// TwinCAT 3 PLC project Main
// ProgramVersion: 3.1.4026.19
// libraries:
//   Tc2_EtherCAT, * (Beckhoff Automation GmbH)
//   Tc2_MC2, * (Beckhoff Automation GmbH)
//   Tc2_Standard, * (Beckhoff Automation GmbH)
//   Tc2_System, * (Beckhoff Automation GmbH)
//   Tc2_Utilities, * (Beckhoff Automation GmbH)
//   Tc3_Database, * (Beckhoff Automation GmbH)
//   Tc3_EventLogger, * (Beckhoff Automation GmbH)
//   Tc3_JsonXml, * (Beckhoff Automation GmbH)
//   Tc3_Module, * (Beckhoff Automation GmbH)
// project tree:
//   DUTs/ ActionMode.TcDUT, MachineState.TcDUT, Sub_Step.TcDUT, TestAction.TcDUT
//   DUTs/IO模組/ IO_In16.TcDUT, IO_Out16.TcDUT
//   DUTs/Jog_STRUCT/ Jog_Laser_Group.TcDUT, Jog_Fx_Group.TcDUT
//   DUTs/加工資料結構/材料加工資訊結構/ tsSteelData.TcDUT
//   DUTs/加工資料結構/工單結構/ WorkOrder_Data.TcDUT
//   DUTs/加工資料結構/雷射加工參數/ LaserParameter_Data.TcDUT
//   DUTs/加工資料結構/雷射加工資料/ LaserProcess_Data.TcDUT
//   DUTs/座標/ XYZ_Point.TcDUT
//   GVLs/ Axis.TcGVL, GrobelVariable.TcGVL, Hmi.TcGVL, Hmi_Web.TcGVL, MaCfg.TcGVL, IO.TcGVL, PosC.TcGVL, ProjectData.TcGVL, RecipeManager.TcRMO (not stored), Safety.TcGVL, SensorTest.TcGVL, AxisTest.TcGVL, SpdC.TcGVL
//   MSG/訊息列表/ MsgBuff.TcGVL
//   MSG/訊息格式/ MsgLevel.TcDUT, MsgStruct.TcDUT, MsgStruct_RAW.TcDUT
//   MSG/通知訊息/ MsgMain.TcPOU, MsgPush.TcPOU, uuidv7_g.TcPOU
//   / PlcTask.TcTTO
//   POUs/ MAIN.TcPOU
//   POUs/功能塊/ ErrorCodeConver.TcPOU, pMsg.TcPOU, RW_Config.TcPOU
//   POUs/功能塊/EtherCat相關/ EtherCat_Driver_Reset.TcPOU, GetEtherSta.TcPOU, EtherCAT_Status.TcPOU
//   POUs/功能塊/Stober驅動/ ReadStoberError.TcPOU, StoberErrorStr.TcPOU
//   POUs/功能塊/字串處理功能塊/字串填充/ FILLSTRING.TcPOU
//   POUs/功能塊/字串處理功能塊/浮點轉字串控制去小數點/ Real2String.TcPOU
//   POUs/功能塊/字串處理功能塊/字串記憶/ WStrMem.TcPOU
//   POUs/功能塊/字串處理功能塊/字串連接/ StrConcat.TcPOU, WStrConcat.TcPOU
//   POUs/功能塊/資料庫 Postgre相關/ ReadSQLData.TcPOU
//   POUs/功能塊/資料庫 Postgre相關/相關結構/取得範圍內的加工資料/ SQL_Get_Payload_Struct.TcDUT
//   POUs/功能塊/資料庫 Postgre相關/相關結構/取得X點/ SQL_GetPosX_Struct.TcDUT
//   POUs/功能塊/資料庫 Postgre相關/相關結構/寫入起始時間/ Payload_Write_Time.TcDUT
//   POUs/功能塊/資料庫 Postgre相關/記錄用/滾輪誤差紀錄/ FxErrPos.TcPOU (not stored), FxErrPos_Struct.TcDUT (not stored)
//   POUs/功能塊/資料庫 Postgre相關/記錄用/程式紀錄/ StepLog_Struct.TcDUT, Step_Log.TcPOU, Step_Log_Clear.TcPOU
//   POUs/動作流程控制/AxisGroup功能塊/ GroupA.TcPOU, GroupB.TcPOU, GroupC.TcPOU, GroupD.TcPOU, GroupFx.TcPOU
//   POUs/動作流程控制/外部輸送滾輪/ ExpConver.TcPOU
//   POUs/安全控制/ MaBaseState.TcPOU
//   POUs/硬體控制/其他控制/按鈕燈/ Button.TcPOU
//   POUs/硬體控制/其他控制/螢幕旋轉/ TurnMonitor.TcPOU
//   POUs/硬體控制/手搖輪/ Jog_MPG.TcPOU
//   POUs/硬體控制/測距感應器/ I_DisSensor.TcIO, OMH555_Decoder.TcPOU, DT80_Decoder.TcPOU, Sensor.TcPOU
//   POUs/硬體控制/軸/ AxisAction.TcPOU, AxisBase.TcPOU, I_Axis.TcIO, MultipleAxisBase.TcPOU, AxisFx.TcPOU
//   POUs/硬體控制/其他控制/三色燈/ LightTower.TcPOU
//   POUs/動作流程控制/ AutoMain.TcPOU
//   POUs/動作流程控制/人機資料轉換/ WebHmi.TcPOU
//   POUs/動作流程控制/測試功能/ Sql_TestData.TcDUT, Sql_TestWriteData.TcDUT, TestActionPou.TcPOU
// real-time tasks:
//   TASK Main_IO_Task: cycle T#2ms, priority 6, ADS port 353
//   TASK PlcTask: cycle T#10ms, priority 14, ADS port 350
//   TASK Conveyor: cycle T#10ms, priority 22, ADS port 355
// motion (NC):
//   TASK NC-Task 1 SAF: cycle T#2ms, priority 4, ADS port 501
//   TASK NC-Task 1 SVB: cycle T#10ms, priority 8, ADS port 511
//   AXIS FX1 (id 1)
//     Dynamic: Acceleration=300, Deceleration=300, Jerk=2000
//     Velo: SlowManual=30, FastManual=300
//     PositionAreaControl: Enable=false
//     OtherSettings: AllowMotionCmdToSlave=true
//     encoder EncType=19
//       EncPara: ScaleFactorNumerator=6.574203208, ScaleFactorDenominator=1048576, Inverse=true, MaxCount=#xffffffff
//     encoder EncId=129, EncType=4
//       EncPara: MaxCount=#xffffffff
//         Inc: RefMode=2
//     encoder EncId=145, EncType=4
//       EncPara: MaxCount=#xffffffff
//         Inc: RefMode=2
//     drive DrvType=16
//       DrvPara: Inverse=true, MaxCount=#xffffffff, DriveControlDWord=#x00020100
//         Analog: TorqueSetpointScale=10, ScaleFactorActTorque=0.1
//         TimeComp: TaskDelayCycles=1
//     controller CtrType=1
//       CtrPara: PriorControlFactor=1
//         PosDiffControl: Enable=false
//         Observer: BandWidth=20
//   AXIS FX2 (id 2)
//     Dynamic: Acceleration=200, Deceleration=200, Jerk=100
//     Velo: FastManual=400, Maximum=600
//     OtherSettings: AllowMotionCmdToSlave=true
//     encoder EncType=19
//       EncPara: ScaleFactorNumerator=6.574203208, ScaleFactorDenominator=1048576, Inverse=true, MaxCount=#xffffffff
//     drive DrvType=16
//       DrvPara: Inverse=true, MaxCount=#xffffffff, DriveControlDWord=#x00020100
//         Analog: TorqueSetpointScale=10, ScaleFactorActTorque=0.1
//         TimeComp: TaskDelayCycles=1
//     controller CtrType=1
//       CtrPara: PriorControlFactor=1
//         Observer: BandWidth=20
//   AXIS AX (id 3)
//     Dynamic: AccelerationMaximum=1000, DecelerationMaximum=1000, Acceleration=1000, Deceleration=1000, Jerk=10000
//     Velo: SlowManual=10, FastManual=50, Maximum=545
//     OtherSettings: AllowMotionCmdToSlave=true, PulseDistancePos=1, PulseDistanceNeg=1
//     encoder EncType=19
//       EncPara: ScaleFactorNumerator=10.6657070589373, ScaleFactorDenominator=1048576, MaxCount=#xffffffff, ReferenceSystem=1
//         SoftEndMinControl: Range=-2
//         SoftEndMaxControl: Range=337
//     drive DrvType=16
//       DrvPara: MaxCount=#xffffffff, DriveControlDWord=#x00020100
//         Analog: VeloReferenz=590, TorqueSetpointScale=10, ScaleFactorActTorque=0.1
//         TimeComp: TaskDelayCycles=1
//     controller CtrType=1
//       CtrPara: PriorControlFactor=1
//         Observer: BandWidth=20
//   AXIS AY (id 4)
//     Dynamic: Acceleration=1000, Deceleration=1000, Jerk=10000
//     Velo: SlowManual=10, FastManual=50, Maximum=545
//     OtherSettings: AllowMotionCmdToSlave=true
//     encoder EncType=19
//       EncPara: ScaleFactorNumerator=10.5986464258042, ScaleFactorDenominator=1048576, Offset=-3.99996967702935, MaxCount=#xffffffff, ReferenceSystem=1
//         SoftEndMinControl: Range=-2
//         SoftEndMaxControl: Range=635.996398925781
//     drive DrvType=16
//       DrvPara: MaxCount=#xffffffff, DriveControlDWord=#x00020100
//         Analog: VeloReferenz=590, TorqueSetpointScale=10, ScaleFactorActTorque=0.1
//         TimeComp: TaskDelayCycles=1
//     controller CtrType=1
//       CtrPara: PriorControlFactor=1
//         Observer: BandWidth=20
//   AXIS AZ1 (id 5)
//     Dynamic: Acceleration=1000, Deceleration=1000, Jerk=10000
//     Velo: SlowManual=10, FastManual=50, Maximum=545
//     OtherSettings: AllowMotionCmdToSlave=true
//     encoder EncType=19
//       EncPara: ScaleFactorNumerator=10.6657070589373, ScaleFactorDenominator=1048576, Inverse=true, MaxCount=#xffffffff, ReferenceSystem=1
//         SoftEndMinControl: Range=-2
//         SoftEndMaxControl: Range=316.997497558594
//     drive DrvType=16
//       DrvPara: Inverse=true, MaxCount=#xffffffff, DriveControlDWord=#x00020100
//         Analog: VeloReferenz=590, TorqueSetpointScale=10, ScaleFactorActTorque=0.1
//         TimeComp: TaskDelayCycles=1
//     controller CtrType=1
//       CtrPara: PriorControlFactor=1
//         Observer: BandWidth=20
//   AXIS AZ2 (id 6)
//     Dynamic: Acceleration=1000, Deceleration=1000, Jerk=10000
//     Velo: SlowManual=10, FastManual=50, Maximum=545
//     OtherSettings: AllowMotionCmdToSlave=true
//     encoder EncType=19
//       EncPara: ScaleFactorNumerator=10.6657070589373, ScaleFactorDenominator=1048576, MaxCount=#xffffffff, ReferenceSystem=1
//     drive DrvType=16
//       DrvPara: MaxCount=#xffffffff, DriveControlDWord=#x00020100
//         Analog: VeloReferenz=590, TorqueSetpointScale=10, ScaleFactorActTorque=0.1
//         TimeComp: TaskDelayCycles=1
//     controller CtrType=1
//       CtrPara: PriorControlFactor=1
//         Observer: BandWidth=20
//   AXIS BX (id 7)
//     Dynamic: Acceleration=1000, Deceleration=1000, Jerk=10000
//     Velo: SlowManual=10, FastManual=50, Maximum=545
//     OtherSettings: AllowMotionCmdToSlave=true
//     encoder EncType=19
//       EncPara: ScaleFactorNumerator=10.6657070589373, ScaleFactorDenominator=1048576, Inverse=true, MaxCount=#xffffffff, ReferenceSystem=1
//         SoftEndMinControl: Range=10
//         SoftEndMaxControl: Range=400
//         Inc: RefSoftSyncMask=#xffffffff
//     drive DrvType=16
//       DrvPara: Inverse=true, MaxCount=#xffffffff, DriveControlDWord=#x00020100
//         Analog: VeloReferenz=590, TorqueSetpointScale=10, ScaleFactorActTorque=0.1
//         TimeComp: TaskDelayCycles=1
//     controller CtrType=1
//       CtrPara: PriorControlFactor=1
//         Observer: BandWidth=20
//   AXIS BY1 (id 8)
//     Dynamic: Acceleration=1000, Deceleration=1000, Jerk=10000
//     Velo: SlowManual=10, FastManual=50, Maximum=545
//     BacklashCompensation: Range=0.05
//     OtherSettings: AllowMotionCmdToSlave=true
//     encoder EncType=19
//       EncPara: ScaleFactorNumerator=10.6657070589373, ScaleFactorDenominator=1048576, Inverse=true, MaxCount=#xffffffff, ReferenceSystem=1
//         SoftEndMinControl: Range=-2
//         SoftEndMaxControl: Range=1405
//     drive DrvType=16
//       DrvPara: Inverse=true, MaxCount=#xffffffff, DriveControlDWord=#x00020100
//         Analog: VeloReferenz=590, TorqueSetpointScale=10, ScaleFactorActTorque=0.1
//         TimeComp: TaskDelayCycles=1
//     controller CtrType=1
//       CtrPara: PriorControlFactor=1
//         Observer: BandWidth=20
//   AXIS BY2 (id 9)
//     Dynamic: Acceleration=1000, Deceleration=1000, Jerk=10000
//     Velo: SlowManual=10, FastManual=50, Maximum=545
//     OtherSettings: ErrorReactionDelay=0.05, AllowMotionCmdToSlave=true
//     encoder EncType=19
//       EncPara: ScaleFactorNumerator=10.6657070589373, ScaleFactorDenominator=1048576, MaxCount=#xffffffff, ReferenceSystem=1
//     drive DrvType=16
//       DrvPara: MaxCount=#xffffffff, DriveControlDWord=#x00020100
//         Analog: VeloReferenz=590, TorqueSetpointScale=10, ScaleFactorActTorque=0.1
//         TimeComp: TaskDelayCycles=1
//     controller CtrType=1
//       CtrPara: PriorControlFactor=1
//         Observer: BandWidth=20
//   AXIS BZ (id 10)
//     Dynamic: Acceleration=1000, Deceleration=1000, Jerk=10000
//     Velo: SlowManual=10, FastManual=50, Maximum=545
//     OtherSettings: AllowMotionCmdToSlave=true
//     encoder EncType=19
//       EncPara: ScaleFactorNumerator=10.6657070589373, ScaleFactorDenominator=1048576, Inverse=true, MaxCount=#xffffffff, ReferenceSystem=1
//         SoftEndMinControl: Range=-2
//         SoftEndMaxControl: Range=601.999633789063
//     drive DrvType=16
//       DrvPara: Inverse=true, MaxCount=#xffffffff, DriveControlDWord=#x00020100
//         Analog: VeloReferenz=590, TorqueSetpointScale=10, ScaleFactorActTorque=0.1
//         TimeComp: TaskDelayCycles=1
//     controller CtrType=1
//       CtrPara: PriorControlFactor=1
//         Observer: BandWidth=20
//   AXIS CX (id 11)
//     Dynamic: Acceleration=1000, Deceleration=1000, Jerk=10000
//     Velo: SlowManual=10, FastManual=50, Maximum=545
//     OtherSettings: AllowMotionCmdToSlave=true
//     encoder EncType=19
//       EncPara: ScaleFactorNumerator=10.6657070589373, ScaleFactorDenominator=1048576, Inverse=true, MaxCount=#xffffffff, ReferenceSystem=1
//         SoftEndMinControl: Range=-2
//         SoftEndMaxControl: Range=317.003509521484
//     drive DrvType=16
//       DrvPara: Inverse=true, MaxCount=#xffffffff, DriveControlDWord=#x00020100
//         Analog: VeloReferenz=590, TorqueSetpointScale=10, ScaleFactorActTorque=0.1
//         TimeComp: TaskDelayCycles=1
//     controller CtrType=1
//       CtrPara: PriorControlFactor=1
//         Observer: BandWidth=20
//   AXIS CY (id 12)
//     Dynamic: Acceleration=1000, Deceleration=1000, Jerk=10000
//     Velo: SlowManual=10, FastManual=50, Maximum=545
//     OtherSettings: AllowMotionCmdToSlave=true
//     encoder EncType=19
//       EncPara: ScaleFactorNumerator=10.6657070589373, ScaleFactorDenominator=1048576, Inverse=true, MaxCount=#xffffffff, ReferenceSystem=1
//         SoftEndMinControl: Range=-2
//         SoftEndMaxControl: Range=623.000061035156
//     drive DrvType=16
//       DrvPara: Inverse=true, MaxCount=#xffffffff, DriveControlDWord=#x00020100
//         Analog: VeloReferenz=590, TorqueSetpointScale=10, ScaleFactorActTorque=0.1
//         TimeComp: TaskDelayCycles=1
//     controller CtrType=1
//       CtrPara: PriorControlFactor=1
//         Observer: BandWidth=20
//   AXIS CZ1 (id 13)
//     Dynamic: Acceleration=1000, Deceleration=1000, Jerk=10000
//     Velo: SlowManual=10, FastManual=50, Maximum=545
//     OtherSettings: AllowMotionCmdToSlave=true
//     encoder EncType=19
//       EncPara: ScaleFactorNumerator=10.6657070589373, ScaleFactorDenominator=1048576, EncMode=3, MaxCount=#xffffffff, ReferenceSystem=1
//         SoftEndMinControl: Range=-2
//         SoftEndMaxControl: Range=1231.99340820313
//     drive DrvType=16
//       DrvPara: MaxCount=#xffffffff, DriveControlDWord=#x00020100
//         Analog: VeloReferenz=590, TorqueSetpointScale=10, ScaleFactorActTorque=0.1
//         TimeComp: TaskDelayCycles=1
//     controller CtrType=1
//       CtrPara: PriorControlFactor=1
//         Observer: BandWidth=20
//   AXIS CZ2 (id 14)
//     Dynamic: Acceleration=1000, Deceleration=1000, Jerk=10000
//     Velo: SlowManual=10, FastManual=50, Maximum=545
//     OtherSettings: AllowMotionCmdToSlave=true
//     encoder EncType=19
//       EncPara: ScaleFactorNumerator=10.6657070589373, ScaleFactorDenominator=1048576, Inverse=true, MaxCount=#xffffffff, ReferenceSystem=1
//     drive DrvType=16
//       DrvPara: Inverse=true, MaxCount=#xffffffff, DriveControlDWord=#x00020100
//         Analog: VeloReferenz=590, TorqueSetpointScale=10, ScaleFactorActTorque=0.1
//         TimeComp: TaskDelayCycles=1
//     controller CtrType=1
//       CtrPara: PriorControlFactor=1
//         Observer: BandWidth=20
//   AXIS DX (id 15)
//     Dynamic: Acceleration=1000, Deceleration=1000, Jerk=10000
//     Velo: SlowManual=10, FastManual=50, Maximum=545
//     OtherSettings: AllowMotionCmdToSlave=true
//     encoder EncType=19
//       EncPara: ScaleFactorNumerator=10.6657070589373, ScaleFactorDenominator=1048576, Offset=-2.99948538910209, Inverse=true, MaxCount=#xffffffff, ReferenceSystem=1
//         SoftEndMinControl: Range=-2
//         SoftEndMaxControl: Range=321.993438720703
//     drive DrvType=16
//       DrvPara: Inverse=true, MaxCount=#xffffffff, DriveControlDWord=#x00020100
//         Analog: VeloReferenz=590, TorqueSetpointScale=10, ScaleFactorActTorque=0.1
//         TimeComp: TaskDelayCycles=1
//     controller CtrType=1
//       CtrPara: PriorControlFactor=1
//         Observer: BandWidth=20
//   AXIS DY (id 16)
//     Dynamic: Acceleration=1000, Deceleration=1000, Jerk=10000
//     Velo: SlowManual=10, FastManual=50, Maximum=545
//     OtherSettings: AllowMotionCmdToSlave=true
//     encoder EncType=19
//       EncPara: ScaleFactorNumerator=10.6657070589373, ScaleFactorDenominator=1048576, MaxCount=#xffffffff, ReferenceSystem=1
//         SoftEndMinControl: Range=-2
//         SoftEndMaxControl: Range=1272
//     drive DrvType=16
//       DrvPara: MaxCount=#xffffffff, DriveControlDWord=#x00020100
//         Analog: VeloReferenz=590, TorqueSetpointScale=10, ScaleFactorActTorque=0.1
//         TimeComp: TaskDelayCycles=1
//     controller CtrType=1
//       CtrPara: PriorControlFactor=1
//         Observer: BandWidth=20
//   AXIS DZ (id 17)
//     Dynamic: Acceleration=1000, Deceleration=1000, Jerk=10000
//     Velo: SlowManual=10, FastManual=50, Maximum=545
//     OtherSettings: AllowMotionCmdToSlave=true
//     encoder EncType=19
//       EncPara: ScaleFactorNumerator=10.6657070589373, ScaleFactorDenominator=1048576, MaxCount=#xffffffff, ReferenceSystem=1
//         SoftEndMinControl: Range=-2
//         SoftEndMaxControl: Range=306.999847412109
//     drive DrvType=16
//       DrvPara: MaxCount=#xffffffff, DriveControlDWord=#x00020100
//         Analog: VeloReferenz=590, TorqueSetpointScale=10, ScaleFactorActTorque=0.1
//         TimeComp: TaskDelayCycles=1
//     controller CtrType=1
//       CtrPara: PriorControlFactor=1
//         Observer: BandWidth=20
//   AXIS MPG (id 18)
//     Dynamic: AccelerationMaximum=50, DecelerationMaximum=50
//     PositionAreaControl: Enable=false
//     TargetPosControl: Enable=false
//     OtherSettings: AllowMotionCmdToSlave=true
//     encoder EncType=4
//       EncPara: ScaleFactorNumerator=1, ModuloFactor=100, EncMode=3, MaxCount=#xffffffff
//         FilterTime: TPos=0.1, TVelo=0, TAcc=0
//         SoftEndMinControl: Range=-3
//         SoftEndMaxControl: Range=-99999
//         ActPosCorrection: Time=0.05
//     drive DrvType=5
//       Analog: VeloReferenz=500, TorqueSetpointScale=10, ScaleFactorActTorque=0.1
//       TimeComp: TaskDelayCycles=1
//     controller CtrType=1
//       CtrPara: PriorControlFactor=1
//         PosDiffControl: Enable=false
//         Observer: BandWidth=20
//   AXIS 轴 19 (id 19)
//     Dynamic: Acceleration=1000, Deceleration=1000, Jerk=5000
//     Velo: SlowManual=10, FastManual=120
//     OtherSettings: AllowMotionCmdToSlave=true
//     encoder EncType=19
//       EncPara: ScaleFactorNumerator=20, ScaleFactorDenominator=10000, ModuloFactor=20, MaxCount=#xffffffff
//     drive DrvType=16
//       DrvPara: MaxCount=#xffffffff, DriveControlDWord=#x00020100
//         Analog: TorqueSetpointScale=10, ScaleFactorActTorque=0.1
//         TimeComp: TaskDelayCycles=1
//     controller CtrType=1
//       CtrPara: PriorControlFactor=1
//         PosDiffControl: Enable=false
//         Observer: BandWidth=20
// I/O:
//   DEVICE Device 1 (EtherCAT), AmsNetId 0.0.0.0.2.1
//     Term 1 (EK1200) [EK1200-5000 EtherCAT Power supply (2A E-Bus)]
//       Term 2 (EL1409) [EL1409 16Ch. Dig. Input 24V, 3ms]
//       Term 3 (EL1409) [EL1409 16Ch. Dig. Input 24V, 3ms]
//       Term 4 (EL1409) [EL1409 16Ch. Dig. Input 24V, 3ms]
//       Term 5 (EL1409) [EL1409 16Ch. Dig. Input 24V, 3ms]
//       Term 6 (EL1409) [EL1409 16Ch. Dig. Input 24V, 3ms]
//       Term 7 (EL1409) [EL1409 16Ch. Dig. Input 24V, 3ms]
//       Term 8 (EL2409) [EL2409 16Ch. Dig. Output 24V, 0.5A]
//       Term 9 (EL2409) [EL2409 16Ch. Dig. Output 24V, 0.5A]
//       Term 10 (EL2409) [EL2409 16Ch. Dig. Output 24V, 0.5A]
//       Term 11 (EL9011) [EL9011 End Terminal]
//   DEVICE Device 2 (EtherCAT), AmsNetId 0.0.0.0.3.1
//     Box 1 (AMAX-4870) [AMAX-4870 4x EtherCAT junction]
//       Box 2 (AMAX-4870) [AMAX-4870 4x EtherCAT junction]
//         Box 3 (AMAX-4870) [AMAX-4870 4x EtherCAT junction]
//           Box 4 (AMAX-4870) [AMAX-4870 4x EtherCAT junction]
//             Term 26 (EK1100) [EK1100 EtherCAT Coupler (2A E-Bus)]
//               Term 27 (EL5102) [EL5102 2Ch. Inc. Encoder 5V (RS422,TTL)] // EL5102 // 修改模組特殊參數時必須先填入 (ASCII:user) Code word(f008) : 75 73 65 72 // 第1組編碼器設定 // 反轉編碼器 : true Reversion of rotation(8000:0E) : 01 // 設定編碼器電壓 : 24V Supply voltage(8001:17) : 0x240 // 計數器上限 : (4,294,967,295) Limit counter value(8001:1A) : FFFFFFFF // 訊號類型 (422+AB相) Counter mode (8001:1D) : 0 // 第2組編碼器設定 // 反轉編碼器 : true Reversion of rotation(8010:0E) : 01 // 設定編碼器電壓 : 24V Supply voltage(8011:17) : 0x240 // 計數器上限 : (4,294,967,295) Limit counter value(8011:1A) : FFFFFFFF // 訊號類型 (422+AB相) Counter mode (8011:1D) : 0
//               Term 28 (EL5102) [EL5102 2Ch. Inc. Encoder 5V (RS422,TTL)] // EL5102 // 修改模組特殊參數時必須先填入 (ASCII:user) Code word(f008) : 75 73 65 72 // 第1組編碼器設定 // 反轉編碼器 : true Reversion of rotation(8000:0E) : 01 // 設定編碼器電壓 : 24V Supply voltage(8001:17) : 0x240 // 計數器上限 : (4,294,967,295) Limit counter value(8001:1A) : FFFFFFFF // 訊號類型 (422+AB相) Counter mode (8001:1D) : 0 // 第2組編碼器設定 // 反轉編碼器 : true Reversion of rotation(8010:0E) : 01 // 設定編碼器電壓 : 24V Supply voltage(8011:17) : 0x240 // 計數器上限 : (4,294,967,295) Limit counter value(8011:1A) : FFFFFFFF // 訊號類型 (422+AB相) Counter mode (8011:1D) : 0
//               Term 29 (EL5102) [EL5102 2Ch. Inc. Encoder 5V (RS422,TTL)] // // 修改模組特殊參數時必須先填入 (ASCII:user) Code word(f008) : 75 73 65 72
//               Term 30 (EL5102) [EL5102 2Ch. Inc. Encoder 5V (RS422,TTL)] // CH1: 測常盤 出口 CH2: 測常盤 入口
//               Term 30 (EL9011) [EL9011 End Terminal]
//           Box 5 (SI6/SC6 2Ax) [SI6/SC6 2Ax]
//             modules: Module 1 (CiA), Module 2 (CiA)
//           Box 6 (SI6/SC6 2Ax) [SI6/SC6 2Ax]
//             modules: Module 1 (CiA), Module 2 (CiA)
//           Box 7 (SI6/SC6 2Ax) [SI6/SC6 2Ax]
//             modules: Module 1 (CiA), Module 2 (CiA)
//           Box 8 (SI6/SC6 2Ax) [SI6/SC6 2Ax]
//             modules: Module 1 (CiA), Module 2 (CiA)
//           Box 9 (SI6/SC6 2Ax) [SI6/SC6 2Ax]
//             modules: Module 1 (CiA), Module 2 (CiA)
//           Box 10 (SI6/SC6 2Ax) [SI6/SC6 2Ax]
//             modules: Module 1 (CiA), Module 2 (CiA)
//           Box 11 (SI6/SC6 2Ax) [SI6/SC6 2Ax]
//             modules: Module 1 (CiA), Module 2 (CiA)
//           Box 12 (SI6/SC6 2Ax) [SI6/SC6 2Ax]
//             modules: Module 1 (CiA), Module 2 (CiA)
//           Box 13 (SI6/SC6 2Ax) [SI6/SC6 2Ax]
//             modules: Module 1 (CiA), Module 2 (CiA)
//         Box 14 (54632) [IMPACT67 Pro EC DIO8 IOL8 M12L 5P]
//           modules: Module 1 (IOL_4/4_I/O-Bytes), Module 2 (IOL_4/4_I/O-Bytes), Module 3 (IOL_4/4_I/O-Bytes), Module 4 (IOL_4/4_I/O-Bytes), Module 5 (Digital_IN), Module 6 (Digital_IN), Module 7 (Digital_IN), Module 8 (IOL_8/8_I/O-Bytes)
//       Box 51 (BL 570)
//       驱动器 71 (CL3-E57H) [CL3-E57H]
// variable links:
//   NC-Task 1 SAF/Axes/AX <-> Device 2 (EtherCAT)/Box 1 (AMAX-4870)/Box 2 (AMAX-4870)/Box 3 (AMAX-4870)/Box 6 (SI6/SC6 2Ax)
//     Drive/Inputs/In/nDataIn1 <-> Module 1 (CiA)/Axis A to Master/1.A632 Following error actual value
//     Drive/Inputs/In/nDataIn3[0] <-> Module 1 (CiA)/Axis A to Master/1.A564 Torque actual value
//     Drive/Inputs/In/nDcOutputTime <-> InfoData/DcOutputShift
//     Drive/Inputs/In/nState1 <-> Module 1 (CiA)/Axis A to Master/1.A516 Statusword
//     Drive/Inputs/In/nState2 <-> Module 1 (CiA)/Axis A to Master/1.A516 Statusword @bit 8
//     Drive/Inputs/In/nState4 @bit 1 <-> WcState/InputToggle
//     Drive/Inputs/In/nState4 <-> WcState/WcState
//     Drive/Inputs/In/nState5 <-> Module 1 (CiA)/Axis A to Master/1.A542 Modes of operation display
//     Drive/Outputs/Out/nCtrl1 <-> Module 1 (CiA)/Axis A to Slave/1.A515 Controlword
//     Drive/Outputs/Out/nCtrl2 <-> Module 1 (CiA)/Axis A to Slave/1.A515 Controlword @bit 8
//     Drive/Outputs/Out/nCtrl5 <-> Module 1 (CiA)/Axis A to Slave/1.A541 Modes of operation
//     Drive/Outputs/Out/nDataOut1 <-> Module 1 (CiA)/Axis A to Slave/1.A567 Target position
//     Drive/Outputs/Out/nDataOut2 <-> Module 1 (CiA)/Axis A to Slave/1.A638 Target velocity
//     Drive/Outputs/Out/nDataOut3[0] <-> Module 1 (CiA)/Axis A to Slave/1.A593 Torque offset
//     Drive/Outputs/Out/nDataOut4[0] <-> Module 1 (CiA)/Axis A to Slave/1.A558 Target torque
//     Enc/Inputs/In/nDataIn1 <-> Module 1 (CiA)/Axis A to Master/1.A545 Position actual value
//     Enc/Inputs/In/nDataIn7 <-> Module 1 (CiA)/Axis A to Master/1.A553 Velocity actual value
//     Enc/Inputs/In/nDcInputTime <-> InfoData/DcInputShift
//     Enc/Inputs/In/nState4 @bit 1 <-> WcState/InputToggle
//     Enc/Inputs/In/nState4 <-> WcState/WcState
//   NC-Task 1 SAF/Axes/AY <-> Device 2 (EtherCAT)/Box 1 (AMAX-4870)/Box 2 (AMAX-4870)/Box 3 (AMAX-4870)/Box 6 (SI6/SC6 2Ax)
//     Drive/Inputs/In/nDataIn1 <-> Module 2 (CiA)/Axis B to Master/2.A632 Following error actual value
//     Drive/Inputs/In/nDataIn3[0] <-> Module 2 (CiA)/Axis B to Master/2.A564 Torque actual value
//     Drive/Inputs/In/nDcOutputTime <-> InfoData/DcOutputShift
//     Drive/Inputs/In/nState1 <-> Module 2 (CiA)/Axis B to Master/2.A516 Statusword
//     Drive/Inputs/In/nState2 <-> Module 2 (CiA)/Axis B to Master/2.A516 Statusword @bit 8
//     Drive/Inputs/In/nState4 @bit 1 <-> WcState/InputToggle
//     Drive/Inputs/In/nState4 <-> WcState/WcState
//     Drive/Inputs/In/nState5 <-> Module 2 (CiA)/Axis B to Master/2.A542 Modes of operation display
//     Drive/Outputs/Out/nCtrl1 <-> Module 2 (CiA)/Axis B to Slave/2.A515 Controlword
//     Drive/Outputs/Out/nCtrl2 <-> Module 2 (CiA)/Axis B to Slave/2.A515 Controlword @bit 8
//     Drive/Outputs/Out/nCtrl5 <-> Module 2 (CiA)/Axis B to Slave/2.A541 Modes of operation
//     Drive/Outputs/Out/nDataOut1 <-> Module 2 (CiA)/Axis B to Slave/2.A567 Target position
//     Drive/Outputs/Out/nDataOut2 <-> Module 2 (CiA)/Axis B to Slave/2.A638 Target velocity
//     Drive/Outputs/Out/nDataOut3[0] <-> Module 2 (CiA)/Axis B to Slave/2.A593 Torque offset
//     Drive/Outputs/Out/nDataOut4[0] <-> Module 2 (CiA)/Axis B to Slave/2.A558 Target torque
//     Enc/Inputs/In/nDataIn1 <-> Module 2 (CiA)/Axis B to Master/2.A545 Position actual value
//     Enc/Inputs/In/nDataIn7 <-> Module 2 (CiA)/Axis B to Master/2.A553 Velocity actual value
//     Enc/Inputs/In/nDcInputTime <-> InfoData/DcInputShift
//     Enc/Inputs/In/nState4 @bit 1 <-> WcState/InputToggle
//     Enc/Inputs/In/nState4 <-> WcState/WcState
//   NC-Task 1 SAF/Axes/AZ1 <-> Device 2 (EtherCAT)/Box 1 (AMAX-4870)/Box 2 (AMAX-4870)/Box 3 (AMAX-4870)/Box 7 (SI6/SC6 2Ax)
//     Drive/Inputs/In/nDataIn1 <-> Module 1 (CiA)/Axis A to Master/1.A632 Following error actual value
//     Drive/Inputs/In/nDataIn3[0] <-> Module 1 (CiA)/Axis A to Master/1.A564 Torque actual value
//     Drive/Inputs/In/nDcOutputTime <-> InfoData/DcOutputShift
//     Drive/Inputs/In/nState1 <-> Module 1 (CiA)/Axis A to Master/1.A516 Statusword
//     Drive/Inputs/In/nState2 <-> Module 1 (CiA)/Axis A to Master/1.A516 Statusword @bit 8
//     Drive/Inputs/In/nState4 @bit 1 <-> WcState/InputToggle
//     Drive/Inputs/In/nState4 <-> WcState/WcState
//     Drive/Inputs/In/nState5 <-> Module 1 (CiA)/Axis A to Master/1.A542 Modes of operation display
//     Drive/Outputs/Out/nCtrl1 <-> Module 1 (CiA)/Axis A to Slave/1.A515 Controlword
//     Drive/Outputs/Out/nCtrl2 <-> Module 1 (CiA)/Axis A to Slave/1.A515 Controlword @bit 8
//     Drive/Outputs/Out/nCtrl5 <-> Module 1 (CiA)/Axis A to Slave/1.A541 Modes of operation
//     Drive/Outputs/Out/nDataOut1 <-> Module 1 (CiA)/Axis A to Slave/1.A567 Target position
//     Drive/Outputs/Out/nDataOut2 <-> Module 1 (CiA)/Axis A to Slave/1.A638 Target velocity
//     Drive/Outputs/Out/nDataOut3[0] <-> Module 1 (CiA)/Axis A to Slave/1.A593 Torque offset
//     Drive/Outputs/Out/nDataOut4[0] <-> Module 1 (CiA)/Axis A to Slave/1.A558 Target torque
//     Enc/Inputs/In/nDataIn1 <-> Module 1 (CiA)/Axis A to Master/1.A545 Position actual value
//     Enc/Inputs/In/nDataIn7 <-> Module 1 (CiA)/Axis A to Master/1.A553 Velocity actual value
//     Enc/Inputs/In/nDcInputTime <-> InfoData/DcInputShift
//     Enc/Inputs/In/nState4 @bit 1 <-> WcState/InputToggle
//     Enc/Inputs/In/nState4 <-> WcState/WcState
//   NC-Task 1 SAF/Axes/AZ2 <-> Device 2 (EtherCAT)/Box 1 (AMAX-4870)/Box 2 (AMAX-4870)/Box 3 (AMAX-4870)/Box 7 (SI6/SC6 2Ax)
//     Drive/Inputs/In/nDataIn1 <-> Module 2 (CiA)/Axis B to Master/2.A632 Following error actual value
//     Drive/Inputs/In/nDataIn3[0] <-> Module 2 (CiA)/Axis B to Master/2.A564 Torque actual value
//     Drive/Inputs/In/nDcOutputTime <-> InfoData/DcOutputShift
//     Drive/Inputs/In/nState1 <-> Module 2 (CiA)/Axis B to Master/2.A516 Statusword
//     Drive/Inputs/In/nState2 <-> Module 2 (CiA)/Axis B to Master/2.A516 Statusword @bit 8
//     Drive/Inputs/In/nState4 @bit 1 <-> WcState/InputToggle
//     Drive/Inputs/In/nState4 <-> WcState/WcState
//     Drive/Inputs/In/nState5 <-> Module 2 (CiA)/Axis B to Master/2.A542 Modes of operation display
//     Drive/Outputs/Out/nCtrl1 <-> Module 2 (CiA)/Axis B to Slave/2.A515 Controlword
//     Drive/Outputs/Out/nCtrl2 <-> Module 2 (CiA)/Axis B to Slave/2.A515 Controlword @bit 8
//     Drive/Outputs/Out/nCtrl5 <-> Module 2 (CiA)/Axis B to Slave/2.A541 Modes of operation
//     Drive/Outputs/Out/nDataOut1 <-> Module 2 (CiA)/Axis B to Slave/2.A567 Target position
//     Drive/Outputs/Out/nDataOut2 <-> Module 2 (CiA)/Axis B to Slave/2.A638 Target velocity
//     Drive/Outputs/Out/nDataOut3[0] <-> Module 2 (CiA)/Axis B to Slave/2.A593 Torque offset
//     Drive/Outputs/Out/nDataOut4[0] <-> Module 2 (CiA)/Axis B to Slave/2.A558 Target torque
//     Enc/Inputs/In/nDataIn1 <-> Module 2 (CiA)/Axis B to Master/2.A545 Position actual value
//     Enc/Inputs/In/nDataIn7 <-> Module 2 (CiA)/Axis B to Master/2.A553 Velocity actual value
//     Enc/Inputs/In/nDcInputTime <-> InfoData/DcInputShift
//     Enc/Inputs/In/nState4 @bit 1 <-> WcState/InputToggle
//     Enc/Inputs/In/nState4 <-> WcState/WcState
//   NC-Task 1 SAF/Axes/BX <-> Device 2 (EtherCAT)/Box 1 (AMAX-4870)/Box 2 (AMAX-4870)/Box 3 (AMAX-4870)/Box 8 (SI6/SC6 2Ax)
//     Drive/Inputs/In/nDataIn1 <-> Module 1 (CiA)/Axis A to Master/1.A632 Following error actual value
//     Drive/Inputs/In/nDataIn3[0] <-> Module 1 (CiA)/Axis A to Master/1.A564 Torque actual value
//     Drive/Inputs/In/nDcOutputTime <-> InfoData/DcOutputShift
//     Drive/Inputs/In/nState1 <-> Module 1 (CiA)/Axis A to Master/1.A516 Statusword
//     Drive/Inputs/In/nState2 <-> Module 1 (CiA)/Axis A to Master/1.A516 Statusword @bit 8
//     Drive/Inputs/In/nState4 @bit 1 <-> WcState/InputToggle
//     Drive/Inputs/In/nState4 <-> WcState/WcState
//     Drive/Inputs/In/nState5 <-> Module 1 (CiA)/Axis A to Master/1.A542 Modes of operation display
//     Drive/Outputs/Out/nCtrl1 <-> Module 1 (CiA)/Axis A to Slave/1.A515 Controlword
//     Drive/Outputs/Out/nCtrl2 <-> Module 1 (CiA)/Axis A to Slave/1.A515 Controlword @bit 8
//     Drive/Outputs/Out/nCtrl5 <-> Module 1 (CiA)/Axis A to Slave/1.A541 Modes of operation
//     Drive/Outputs/Out/nDataOut1 <-> Module 1 (CiA)/Axis A to Slave/1.A567 Target position
//     Drive/Outputs/Out/nDataOut2 <-> Module 1 (CiA)/Axis A to Slave/1.A638 Target velocity
//     Drive/Outputs/Out/nDataOut3[0] <-> Module 1 (CiA)/Axis A to Slave/1.A593 Torque offset
//     Drive/Outputs/Out/nDataOut4[0] <-> Module 1 (CiA)/Axis A to Slave/1.A558 Target torque
//     Enc/Inputs/In/nDataIn1 <-> Module 1 (CiA)/Axis A to Master/1.A545 Position actual value
//     Enc/Inputs/In/nDataIn7 <-> Module 1 (CiA)/Axis A to Master/1.A553 Velocity actual value
//     Enc/Inputs/In/nDcInputTime <-> InfoData/DcInputShift
//     Enc/Inputs/In/nState4 @bit 1 <-> WcState/InputToggle
//     Enc/Inputs/In/nState4 <-> WcState/WcState
//   NC-Task 1 SAF/Axes/BY1 <-> Device 2 (EtherCAT)/Box 1 (AMAX-4870)/Box 2 (AMAX-4870)/Box 3 (AMAX-4870)/Box 9 (SI6/SC6 2Ax)
//     Drive/Inputs/In/nDataIn1 <-> Module 1 (CiA)/Axis A to Master/1.A632 Following error actual value
//     Drive/Inputs/In/nDataIn3[0] <-> Module 1 (CiA)/Axis A to Master/1.A564 Torque actual value
//     Drive/Inputs/In/nDcOutputTime <-> InfoData/DcOutputShift
//     Drive/Inputs/In/nState1 <-> Module 1 (CiA)/Axis A to Master/1.A516 Statusword
//     Drive/Inputs/In/nState2 <-> Module 1 (CiA)/Axis A to Master/1.A516 Statusword @bit 8
//     Drive/Inputs/In/nState4 @bit 1 <-> WcState/InputToggle
//     Drive/Inputs/In/nState4 <-> WcState/WcState
//     Drive/Inputs/In/nState5 <-> Module 1 (CiA)/Axis A to Master/1.A542 Modes of operation display
//     Drive/Outputs/Out/nCtrl1 <-> Module 1 (CiA)/Axis A to Slave/1.A515 Controlword
//     Drive/Outputs/Out/nCtrl2 <-> Module 1 (CiA)/Axis A to Slave/1.A515 Controlword @bit 8
//     Drive/Outputs/Out/nCtrl5 <-> Module 1 (CiA)/Axis A to Slave/1.A541 Modes of operation
//     Drive/Outputs/Out/nDataOut1 <-> Module 1 (CiA)/Axis A to Slave/1.A567 Target position
//     Drive/Outputs/Out/nDataOut2 <-> Module 1 (CiA)/Axis A to Slave/1.A638 Target velocity
//     Drive/Outputs/Out/nDataOut3[0] <-> Module 1 (CiA)/Axis A to Slave/1.A593 Torque offset
//     Drive/Outputs/Out/nDataOut4[0] <-> Module 1 (CiA)/Axis A to Slave/1.A558 Target torque
//     Enc/Inputs/In/nDataIn1 <-> Module 1 (CiA)/Axis A to Master/1.A545 Position actual value
//     Enc/Inputs/In/nDataIn7 <-> Module 1 (CiA)/Axis A to Master/1.A553 Velocity actual value
//     Enc/Inputs/In/nDcInputTime <-> InfoData/DcInputShift
//     Enc/Inputs/In/nState4 @bit 1 <-> WcState/InputToggle
//     Enc/Inputs/In/nState4 <-> WcState/WcState
//   NC-Task 1 SAF/Axes/BY2 <-> Device 2 (EtherCAT)/Box 1 (AMAX-4870)/Box 2 (AMAX-4870)/Box 3 (AMAX-4870)/Box 9 (SI6/SC6 2Ax)
//     Drive/Inputs/In/nDataIn1 <-> Module 2 (CiA)/Axis B to Master/2.A632 Following error actual value
//     Drive/Inputs/In/nDataIn3[0] <-> Module 2 (CiA)/Axis B to Master/2.A564 Torque actual value
//     Drive/Inputs/In/nDcOutputTime <-> InfoData/DcOutputShift
//     Drive/Inputs/In/nState1 <-> Module 2 (CiA)/Axis B to Master/2.A516 Statusword
//     Drive/Inputs/In/nState2 <-> Module 2 (CiA)/Axis B to Master/2.A516 Statusword @bit 8
//     Drive/Inputs/In/nState4 @bit 1 <-> WcState/InputToggle
//     Drive/Inputs/In/nState4 <-> WcState/WcState
//     Drive/Inputs/In/nState5 <-> Module 2 (CiA)/Axis B to Master/2.A542 Modes of operation display
//     Drive/Outputs/Out/nCtrl1 <-> Module 2 (CiA)/Axis B to Slave/2.A515 Controlword
//     Drive/Outputs/Out/nCtrl2 <-> Module 2 (CiA)/Axis B to Slave/2.A515 Controlword @bit 8
//     Drive/Outputs/Out/nCtrl5 <-> Module 2 (CiA)/Axis B to Slave/2.A541 Modes of operation
//     Drive/Outputs/Out/nDataOut1 <-> Module 2 (CiA)/Axis B to Slave/2.A567 Target position
//     Drive/Outputs/Out/nDataOut2 <-> Module 2 (CiA)/Axis B to Slave/2.A638 Target velocity
//     Drive/Outputs/Out/nDataOut3[0] <-> Module 2 (CiA)/Axis B to Slave/2.A593 Torque offset
//     Drive/Outputs/Out/nDataOut4[0] <-> Module 2 (CiA)/Axis B to Slave/2.A558 Target torque
//     Enc/Inputs/In/nDataIn1 <-> Module 2 (CiA)/Axis B to Master/2.A545 Position actual value
//     Enc/Inputs/In/nDataIn7 <-> Module 2 (CiA)/Axis B to Master/2.A553 Velocity actual value
//     Enc/Inputs/In/nDcInputTime <-> InfoData/DcInputShift
//     Enc/Inputs/In/nState4 @bit 1 <-> WcState/InputToggle
//     Enc/Inputs/In/nState4 <-> WcState/WcState
//   NC-Task 1 SAF/Axes/BZ <-> Device 2 (EtherCAT)/Box 1 (AMAX-4870)/Box 2 (AMAX-4870)/Box 3 (AMAX-4870)/Box 8 (SI6/SC6 2Ax)
//     Drive/Inputs/In/nDataIn1 <-> Module 2 (CiA)/Axis B to Master/2.A632 Following error actual value
//     Drive/Inputs/In/nDataIn3[0] <-> Module 2 (CiA)/Axis B to Master/2.A564 Torque actual value
//     Drive/Inputs/In/nDcOutputTime <-> InfoData/DcOutputShift
//     Drive/Inputs/In/nState1 <-> Module 2 (CiA)/Axis B to Master/2.A516 Statusword
//     Drive/Inputs/In/nState2 <-> Module 2 (CiA)/Axis B to Master/2.A516 Statusword @bit 8
//     Drive/Inputs/In/nState4 @bit 1 <-> WcState/InputToggle
//     Drive/Inputs/In/nState4 <-> WcState/WcState
//     Drive/Inputs/In/nState5 <-> Module 2 (CiA)/Axis B to Master/2.A542 Modes of operation display
//     Drive/Outputs/Out/nCtrl1 <-> Module 2 (CiA)/Axis B to Slave/2.A515 Controlword
//     Drive/Outputs/Out/nCtrl2 <-> Module 2 (CiA)/Axis B to Slave/2.A515 Controlword @bit 8
//     Drive/Outputs/Out/nCtrl5 <-> Module 2 (CiA)/Axis B to Slave/2.A541 Modes of operation
//     Drive/Outputs/Out/nDataOut1 <-> Module 2 (CiA)/Axis B to Slave/2.A567 Target position
//     Drive/Outputs/Out/nDataOut2 <-> Module 2 (CiA)/Axis B to Slave/2.A638 Target velocity
//     Drive/Outputs/Out/nDataOut3[0] <-> Module 2 (CiA)/Axis B to Slave/2.A593 Torque offset
//     Drive/Outputs/Out/nDataOut4[0] <-> Module 2 (CiA)/Axis B to Slave/2.A558 Target torque
//     Enc/Inputs/In/nDataIn1 <-> Module 2 (CiA)/Axis B to Master/2.A545 Position actual value
//     Enc/Inputs/In/nDataIn7 <-> Module 2 (CiA)/Axis B to Master/2.A553 Velocity actual value
//     Enc/Inputs/In/nDcInputTime <-> InfoData/DcInputShift
//     Enc/Inputs/In/nState4 @bit 1 <-> WcState/InputToggle
//     Enc/Inputs/In/nState4 <-> WcState/WcState
//   NC-Task 1 SAF/Axes/CX <-> Device 2 (EtherCAT)/Box 1 (AMAX-4870)/Box 2 (AMAX-4870)/Box 3 (AMAX-4870)/Box 10 (SI6/SC6 2Ax)
//     Drive/Inputs/In/nDataIn1 <-> Module 1 (CiA)/Axis A to Master/1.A632 Following error actual value
//     Drive/Inputs/In/nDataIn3[0] <-> Module 1 (CiA)/Axis A to Master/1.A564 Torque actual value
//     Drive/Inputs/In/nDcOutputTime <-> InfoData/DcOutputShift
//     Drive/Inputs/In/nState1 <-> Module 1 (CiA)/Axis A to Master/1.A516 Statusword
//     Drive/Inputs/In/nState2 <-> Module 1 (CiA)/Axis A to Master/1.A516 Statusword @bit 8
//     Drive/Inputs/In/nState4 @bit 1 <-> WcState/InputToggle
//     Drive/Inputs/In/nState4 <-> WcState/WcState
//     Drive/Inputs/In/nState5 <-> Module 1 (CiA)/Axis A to Master/1.A542 Modes of operation display
//     Drive/Outputs/Out/nCtrl1 <-> Module 1 (CiA)/Axis A to Slave/1.A515 Controlword
//     Drive/Outputs/Out/nCtrl2 <-> Module 1 (CiA)/Axis A to Slave/1.A515 Controlword @bit 8
//     Drive/Outputs/Out/nCtrl5 <-> Module 1 (CiA)/Axis A to Slave/1.A541 Modes of operation
//     Drive/Outputs/Out/nDataOut1 <-> Module 1 (CiA)/Axis A to Slave/1.A567 Target position
//     Drive/Outputs/Out/nDataOut2 <-> Module 1 (CiA)/Axis A to Slave/1.A638 Target velocity
//     Drive/Outputs/Out/nDataOut3[0] <-> Module 1 (CiA)/Axis A to Slave/1.A593 Torque offset
//     Drive/Outputs/Out/nDataOut4[0] <-> Module 1 (CiA)/Axis A to Slave/1.A558 Target torque
//     Enc/Inputs/In/nDataIn1 <-> Module 1 (CiA)/Axis A to Master/1.A545 Position actual value
//     Enc/Inputs/In/nDataIn7 <-> Module 1 (CiA)/Axis A to Master/1.A553 Velocity actual value
//     Enc/Inputs/In/nDcInputTime <-> InfoData/DcInputShift
//     Enc/Inputs/In/nState4 @bit 1 <-> WcState/InputToggle
//     Enc/Inputs/In/nState4 <-> WcState/WcState
//   NC-Task 1 SAF/Axes/CY <-> Device 2 (EtherCAT)/Box 1 (AMAX-4870)/Box 2 (AMAX-4870)/Box 3 (AMAX-4870)/Box 10 (SI6/SC6 2Ax)
//     Drive/Inputs/In/nDataIn1 <-> Module 2 (CiA)/Axis B to Master/2.A632 Following error actual value
//     Drive/Inputs/In/nDataIn3[0] <-> Module 2 (CiA)/Axis B to Master/2.A564 Torque actual value
//     Drive/Inputs/In/nDcOutputTime <-> InfoData/DcOutputShift
//     Drive/Inputs/In/nState1 <-> Module 2 (CiA)/Axis B to Master/2.A516 Statusword
//     Drive/Inputs/In/nState2 <-> Module 2 (CiA)/Axis B to Master/2.A516 Statusword @bit 8
//     Drive/Inputs/In/nState4 @bit 1 <-> WcState/InputToggle
//     Drive/Inputs/In/nState4 <-> WcState/WcState
//     Drive/Inputs/In/nState5 <-> Module 2 (CiA)/Axis B to Master/2.A542 Modes of operation display
//     Drive/Outputs/Out/nCtrl1 <-> Module 2 (CiA)/Axis B to Slave/2.A515 Controlword
//     Drive/Outputs/Out/nCtrl2 <-> Module 2 (CiA)/Axis B to Slave/2.A515 Controlword @bit 8
//     Drive/Outputs/Out/nCtrl5 <-> Module 2 (CiA)/Axis B to Slave/2.A541 Modes of operation
//     Drive/Outputs/Out/nDataOut1 <-> Module 2 (CiA)/Axis B to Slave/2.A567 Target position
//     Drive/Outputs/Out/nDataOut2 <-> Module 2 (CiA)/Axis B to Slave/2.A638 Target velocity
//     Drive/Outputs/Out/nDataOut3[0] <-> Module 2 (CiA)/Axis B to Slave/2.A593 Torque offset
//     Drive/Outputs/Out/nDataOut4[0] <-> Module 2 (CiA)/Axis B to Slave/2.A558 Target torque
//     Enc/Inputs/In/nDataIn1 <-> Module 2 (CiA)/Axis B to Master/2.A545 Position actual value
//     Enc/Inputs/In/nDataIn7 <-> Module 2 (CiA)/Axis B to Master/2.A553 Velocity actual value
//     Enc/Inputs/In/nDcInputTime <-> InfoData/DcInputShift
//     Enc/Inputs/In/nState4 @bit 1 <-> WcState/InputToggle
//     Enc/Inputs/In/nState4 <-> WcState/WcState
//   NC-Task 1 SAF/Axes/CZ1 <-> Device 2 (EtherCAT)/Box 1 (AMAX-4870)/Box 2 (AMAX-4870)/Box 3 (AMAX-4870)/Box 11 (SI6/SC6 2Ax)
//     Drive/Inputs/In/nDataIn1 <-> Module 1 (CiA)/Axis A to Master/1.A632 Following error actual value
//     Drive/Inputs/In/nDataIn3[0] <-> Module 1 (CiA)/Axis A to Master/1.A564 Torque actual value
//     Drive/Inputs/In/nDcOutputTime <-> InfoData/DcOutputShift
//     Drive/Inputs/In/nState1 <-> Module 1 (CiA)/Axis A to Master/1.A516 Statusword
//     Drive/Inputs/In/nState2 <-> Module 1 (CiA)/Axis A to Master/1.A516 Statusword @bit 8
//     Drive/Inputs/In/nState4 @bit 1 <-> WcState/InputToggle
//     Drive/Inputs/In/nState4 <-> WcState/WcState
//     Drive/Inputs/In/nState5 <-> Module 1 (CiA)/Axis A to Master/1.A542 Modes of operation display
//     Drive/Outputs/Out/nCtrl1 <-> Module 1 (CiA)/Axis A to Slave/1.A515 Controlword
//     Drive/Outputs/Out/nCtrl2 <-> Module 1 (CiA)/Axis A to Slave/1.A515 Controlword @bit 8
//     Drive/Outputs/Out/nCtrl5 <-> Module 1 (CiA)/Axis A to Slave/1.A541 Modes of operation
//     Drive/Outputs/Out/nDataOut1 <-> Module 1 (CiA)/Axis A to Slave/1.A567 Target position
//     Drive/Outputs/Out/nDataOut2 <-> Module 1 (CiA)/Axis A to Slave/1.A638 Target velocity
//     Drive/Outputs/Out/nDataOut3[0] <-> Module 1 (CiA)/Axis A to Slave/1.A593 Torque offset
//     Drive/Outputs/Out/nDataOut4[0] <-> Module 1 (CiA)/Axis A to Slave/1.A558 Target torque
//     Enc/Inputs/In/nDataIn1 <-> Module 1 (CiA)/Axis A to Master/1.A545 Position actual value
//     Enc/Inputs/In/nDataIn7 <-> Module 1 (CiA)/Axis A to Master/1.A553 Velocity actual value
//     Enc/Inputs/In/nDcInputTime <-> InfoData/DcInputShift
//     Enc/Inputs/In/nState4 @bit 1 <-> WcState/InputToggle
//     Enc/Inputs/In/nState4 <-> WcState/WcState
//   NC-Task 1 SAF/Axes/CZ2 <-> Device 2 (EtherCAT)/Box 1 (AMAX-4870)/Box 2 (AMAX-4870)/Box 3 (AMAX-4870)/Box 11 (SI6/SC6 2Ax)
//     Drive/Inputs/In/nDataIn1 <-> Module 2 (CiA)/Axis B to Master/2.A632 Following error actual value
//     Drive/Inputs/In/nDataIn3[0] <-> Module 2 (CiA)/Axis B to Master/2.A564 Torque actual value
//     Drive/Inputs/In/nDcOutputTime <-> InfoData/DcOutputShift
//     Drive/Inputs/In/nState1 <-> Module 2 (CiA)/Axis B to Master/2.A516 Statusword
//     Drive/Inputs/In/nState2 <-> Module 2 (CiA)/Axis B to Master/2.A516 Statusword @bit 8
//     Drive/Inputs/In/nState4 @bit 1 <-> WcState/InputToggle
//     Drive/Inputs/In/nState4 <-> WcState/WcState
//     Drive/Inputs/In/nState5 <-> Module 2 (CiA)/Axis B to Master/2.A542 Modes of operation display
//     Drive/Outputs/Out/nCtrl1 <-> Module 2 (CiA)/Axis B to Slave/2.A515 Controlword
//     Drive/Outputs/Out/nCtrl2 <-> Module 2 (CiA)/Axis B to Slave/2.A515 Controlword @bit 8
//     Drive/Outputs/Out/nCtrl5 <-> Module 2 (CiA)/Axis B to Slave/2.A541 Modes of operation
//     Drive/Outputs/Out/nDataOut1 <-> Module 2 (CiA)/Axis B to Slave/2.A567 Target position
//     Drive/Outputs/Out/nDataOut2 <-> Module 2 (CiA)/Axis B to Slave/2.A638 Target velocity
//     Drive/Outputs/Out/nDataOut3[0] <-> Module 2 (CiA)/Axis B to Slave/2.A593 Torque offset
//     Drive/Outputs/Out/nDataOut4[0] <-> Module 2 (CiA)/Axis B to Slave/2.A558 Target torque
//     Enc/Inputs/In/nDataIn1 <-> Module 2 (CiA)/Axis B to Master/2.A545 Position actual value
//     Enc/Inputs/In/nDataIn7 <-> Module 2 (CiA)/Axis B to Master/2.A553 Velocity actual value
//     Enc/Inputs/In/nDcInputTime <-> InfoData/DcInputShift
//     Enc/Inputs/In/nState4 @bit 1 <-> WcState/InputToggle
//     Enc/Inputs/In/nState4 <-> WcState/WcState
//   NC-Task 1 SAF/Axes/DX <-> Device 2 (EtherCAT)/Box 1 (AMAX-4870)/Box 2 (AMAX-4870)/Box 3 (AMAX-4870)/Box 12 (SI6/SC6 2Ax)
//     Drive/Inputs/In/nDataIn1 <-> Module 2 (CiA)/Axis B to Master/2.A632 Following error actual value
//     Drive/Inputs/In/nDataIn3[0] <-> Module 2 (CiA)/Axis B to Master/2.A564 Torque actual value
//     Drive/Inputs/In/nDcOutputTime <-> InfoData/DcOutputShift
//     Drive/Inputs/In/nState1 <-> Module 2 (CiA)/Axis B to Master/2.A516 Statusword
//     Drive/Inputs/In/nState2 <-> Module 2 (CiA)/Axis B to Master/2.A516 Statusword @bit 8
//     Drive/Inputs/In/nState4 @bit 1 <-> WcState/InputToggle
//     Drive/Inputs/In/nState4 <-> WcState/WcState
//     Drive/Inputs/In/nState5 <-> Module 2 (CiA)/Axis B to Master/2.A542 Modes of operation display
//     Drive/Outputs/Out/nCtrl1 <-> Module 2 (CiA)/Axis B to Slave/2.A515 Controlword
//     Drive/Outputs/Out/nCtrl2 <-> Module 2 (CiA)/Axis B to Slave/2.A515 Controlword @bit 8
//     Drive/Outputs/Out/nCtrl5 <-> Module 2 (CiA)/Axis B to Slave/2.A541 Modes of operation
//     Drive/Outputs/Out/nDataOut1 <-> Module 2 (CiA)/Axis B to Slave/2.A567 Target position
//     Drive/Outputs/Out/nDataOut2 <-> Module 2 (CiA)/Axis B to Slave/2.A638 Target velocity
//     Drive/Outputs/Out/nDataOut3[0] <-> Module 2 (CiA)/Axis B to Slave/2.A593 Torque offset
//     Drive/Outputs/Out/nDataOut4[0] <-> Module 2 (CiA)/Axis B to Slave/2.A558 Target torque
//     Enc/Inputs/In/nDataIn1 <-> Module 2 (CiA)/Axis B to Master/2.A545 Position actual value
//     Enc/Inputs/In/nDataIn7 <-> Module 2 (CiA)/Axis B to Master/2.A553 Velocity actual value
//     Enc/Inputs/In/nDcInputTime <-> InfoData/DcInputShift
//     Enc/Inputs/In/nState4 @bit 1 <-> WcState/InputToggle
//     Enc/Inputs/In/nState4 <-> WcState/WcState
//   NC-Task 1 SAF/Axes/DY <-> Device 2 (EtherCAT)/Box 1 (AMAX-4870)/Box 2 (AMAX-4870)/Box 3 (AMAX-4870)/Box 12 (SI6/SC6 2Ax)
//     Drive/Inputs/In/nDataIn1 <-> Module 1 (CiA)/Axis A to Master/1.A632 Following error actual value
//     Drive/Inputs/In/nDataIn3[0] <-> Module 1 (CiA)/Axis A to Master/1.A564 Torque actual value
//     Drive/Inputs/In/nDcOutputTime <-> InfoData/DcOutputShift
//     Drive/Inputs/In/nState1 <-> Module 1 (CiA)/Axis A to Master/1.A516 Statusword
//     Drive/Inputs/In/nState2 <-> Module 1 (CiA)/Axis A to Master/1.A516 Statusword @bit 8
//     Drive/Inputs/In/nState4 @bit 1 <-> WcState/InputToggle
//     Drive/Inputs/In/nState4 <-> WcState/WcState
//     Drive/Inputs/In/nState5 <-> Module 1 (CiA)/Axis A to Master/1.A542 Modes of operation display
//     Drive/Outputs/Out/nCtrl1 <-> Module 1 (CiA)/Axis A to Slave/1.A515 Controlword
//     Drive/Outputs/Out/nCtrl2 <-> Module 1 (CiA)/Axis A to Slave/1.A515 Controlword @bit 8
//     Drive/Outputs/Out/nCtrl5 <-> Module 1 (CiA)/Axis A to Slave/1.A541 Modes of operation
//     Drive/Outputs/Out/nDataOut1 <-> Module 1 (CiA)/Axis A to Slave/1.A567 Target position
//     Drive/Outputs/Out/nDataOut2 <-> Module 1 (CiA)/Axis A to Slave/1.A638 Target velocity
//     Drive/Outputs/Out/nDataOut3[0] <-> Module 1 (CiA)/Axis A to Slave/1.A593 Torque offset
//     Drive/Outputs/Out/nDataOut4[0] <-> Module 1 (CiA)/Axis A to Slave/1.A558 Target torque
//     Enc/Inputs/In/nDataIn1 <-> Module 1 (CiA)/Axis A to Master/1.A545 Position actual value
//     Enc/Inputs/In/nDataIn7 <-> Module 1 (CiA)/Axis A to Master/1.A553 Velocity actual value
//     Enc/Inputs/In/nDcInputTime <-> InfoData/DcInputShift
//     Enc/Inputs/In/nState4 @bit 1 <-> WcState/InputToggle
//     Enc/Inputs/In/nState4 <-> WcState/WcState
//   NC-Task 1 SAF/Axes/DZ <-> Device 2 (EtherCAT)/Box 1 (AMAX-4870)/Box 2 (AMAX-4870)/Box 3 (AMAX-4870)/Box 13 (SI6/SC6 2Ax)
//     Drive/Inputs/In/nDataIn1 <-> Module 1 (CiA)/Axis A to Master/1.A632 Following error actual value
//     Drive/Inputs/In/nDataIn3[0] <-> Module 1 (CiA)/Axis A to Master/1.A564 Torque actual value
//     Drive/Inputs/In/nDcOutputTime <-> InfoData/DcOutputShift
//     Drive/Inputs/In/nState1 <-> Module 1 (CiA)/Axis A to Master/1.A516 Statusword
//     Drive/Inputs/In/nState2 <-> Module 1 (CiA)/Axis A to Master/1.A516 Statusword @bit 8
//     Drive/Inputs/In/nState4 @bit 1 <-> WcState/InputToggle
//     Drive/Inputs/In/nState4 <-> WcState/WcState
//     Drive/Inputs/In/nState5 <-> Module 1 (CiA)/Axis A to Master/1.A542 Modes of operation display
//     Drive/Outputs/Out/nCtrl1 <-> Module 1 (CiA)/Axis A to Slave/1.A515 Controlword
//     Drive/Outputs/Out/nCtrl2 <-> Module 1 (CiA)/Axis A to Slave/1.A515 Controlword @bit 8
//     Drive/Outputs/Out/nCtrl5 <-> Module 1 (CiA)/Axis A to Slave/1.A541 Modes of operation
//     Drive/Outputs/Out/nDataOut1 <-> Module 1 (CiA)/Axis A to Slave/1.A567 Target position
//     Drive/Outputs/Out/nDataOut2 <-> Module 1 (CiA)/Axis A to Slave/1.A638 Target velocity
//     Drive/Outputs/Out/nDataOut3[0] <-> Module 1 (CiA)/Axis A to Slave/1.A593 Torque offset
//     Drive/Outputs/Out/nDataOut4[0] <-> Module 1 (CiA)/Axis A to Slave/1.A558 Target torque
//     Enc/Inputs/In/nDataIn1 <-> Module 1 (CiA)/Axis A to Master/1.A545 Position actual value
//     Enc/Inputs/In/nDataIn7 <-> Module 1 (CiA)/Axis A to Master/1.A553 Velocity actual value
//     Enc/Inputs/In/nDcInputTime <-> InfoData/DcInputShift
//     Enc/Inputs/In/nState4 @bit 1 <-> WcState/InputToggle
//     Enc/Inputs/In/nState4 <-> WcState/WcState
//   NC-Task 1 SAF/Axes/FX1 <-> Device 2 (EtherCAT)/Box 1 (AMAX-4870)/Box 2 (AMAX-4870)/Box 3 (AMAX-4870)/Box 4 (AMAX-4870)/Term 26 (EK1100)/Term 27 (EL5102)
//     ExpEncA/输入/In/nDataIn1 <-> ENC Status Channel 1/Counter value
//     ExpEncA/输入/In/nDataIn2 <-> ENC Status Channel 1/Latch value
//     ExpEncA/输入/In/nDcInputTime <-> InfoData/DcInputShift
//     ExpEncA/输入/In/nState1 @bit 4 <-> ENC Status Channel 1/Status/Counter overflow
//     ExpEncA/输入/In/nState1 @bit 3 <-> ENC Status Channel 1/Status/Counter underflow
//     ExpEncA/输入/In/nState1 @bit 7 <-> ENC Status Channel 1/Status/Extrapolation stall
//     ExpEncA/输入/In/nState1 <-> ENC Status Channel 1/Status/Latch C valid
//     ExpEncA/输入/In/nState1 @bit 1 <-> ENC Status Channel 1/Status/Latch extern valid
//     ExpEncA/输入/In/nState1 @bit 6 <-> ENC Status Channel 1/Status/Open circuit
//     ExpEncA/输入/In/nState1 @bit 2 <-> ENC Status Channel 1/Status/Set counter done
//     ExpEncA/输入/In/nState1 @bit 5 <-> ENC Status Channel 1/Status/Status of input status
//     ExpEncA/输入/In/nState2 @bit 4 <-> ENC Status Channel 1/Status/Diag
//     ExpEncA/输入/In/nState2 @bit 6 <-> ENC Status Channel 1/Status/Input cycle counter
//     ExpEncA/输入/In/nState2 <-> ENC Status Channel 1/Status/Status of input A
//     ExpEncA/输入/In/nState2 @bit 1 <-> ENC Status Channel 1/Status/Status of input B
//     ExpEncA/输入/In/nState2 @bit 2 <-> ENC Status Channel 1/Status/Status of input C
//     ExpEncA/输入/In/nState2 @bit 3 <-> ENC Status Channel 1/Status/Status of input gate
//     ExpEncA/输入/In/nState2 @bit 5 <-> ENC Status Channel 1/Status/TxPDO State
//     ExpEncA/输入/In/nState3 @bit 4 <-> ENC Status Channel 1/Status/Counter value out of range
//     ExpEncA/输入/In/nState3 @bit 2 <-> ENC Status Channel 1/Status/Direction inversion detected
//     ExpEncA/输入/In/nState3 @bit 1 <-> ENC Status Channel 1/Status/Latch extern 2 valid
//     ExpEncA/输入/In/nState3 <-> ENC Status Channel 1/Status/Software gate valid
//     ExpEncA/输入/In/nState3 @bit 3 <-> ENC Status Channel 1/Status/Status of extern latch
//     ExpEncA/输入/In/nState4 @bit 1 <-> WcState/InputToggle
//     ExpEncA/输入/In/nState4 <-> WcState/WcState
//     ExpEncA/输出/Out/nCtrl1 <-> ENC Control Channel 1/Control/Enable latch C
//     ExpEncA/输出/Out/nCtrl1 @bit 3 <-> ENC Control Channel 1/Control/Enable latch extern on negative edge
//     ExpEncA/输出/Out/nCtrl1 @bit 1 <-> ENC Control Channel 1/Control/Enable latch extern on positive edge
//     ExpEncA/输出/Out/nCtrl1 @bit 2 <-> ENC Control Channel 1/Control/Set counter
//     ExpEncA/输出/Out/nCtrl1 @bit 7 <-> ENC Control Channel 1/Control/Set counter on latch C
//     ExpEncA/输出/Out/nCtrl2 @bit 4 <-> ENC Control Channel 1/Control/Enable latch extern 2 on negative edge
//     ExpEncA/输出/Out/nCtrl2 @bit 3 <-> ENC Control Channel 1/Control/Enable latch extern 2 on positive edge
//     ExpEncA/输出/Out/nCtrl2 @bit 2 <-> ENC Control Channel 1/Control/Set counter on latch extern on negative edge
//     ExpEncA/输出/Out/nCtrl2 @bit 1 <-> ENC Control Channel 1/Control/Set counter on latch extern on positive edge
//     ExpEncA/输出/Out/nCtrl2 <-> ENC Control Channel 1/Control/Set software gate
//     ExpEncA/输出/Out/nDataOut1 <-> ENC Control Channel 1/Set counter value
//     ExpEncB/输入/In/nDataIn1 <-> ENC Status Channel 2/Counter value
//     ExpEncB/输入/In/nDataIn2 <-> ENC Status Channel 2/Latch value
//     ExpEncB/输入/In/nDcInputTime <-> InfoData/DcInputShift
//     ExpEncB/输入/In/nState1 @bit 4 <-> ENC Status Channel 2/Status/Counter overflow
//     ExpEncB/输入/In/nState1 @bit 3 <-> ENC Status Channel 2/Status/Counter underflow
//     ExpEncB/输入/In/nState1 @bit 7 <-> ENC Status Channel 2/Status/Extrapolation stall
//     ExpEncB/输入/In/nState1 <-> ENC Status Channel 2/Status/Latch C valid
//     ExpEncB/输入/In/nState1 @bit 1 <-> ENC Status Channel 2/Status/Latch extern valid
//     ExpEncB/输入/In/nState1 @bit 6 <-> ENC Status Channel 2/Status/Open circuit
//     ExpEncB/输入/In/nState1 @bit 2 <-> ENC Status Channel 2/Status/Set counter done
//     ExpEncB/输入/In/nState1 @bit 5 <-> ENC Status Channel 2/Status/Status of input status
//     ExpEncB/输入/In/nState2 @bit 4 <-> ENC Status Channel 2/Status/Diag
//     ExpEncB/输入/In/nState2 @bit 6 <-> ENC Status Channel 2/Status/Input cycle counter
//     ExpEncB/输入/In/nState2 <-> ENC Status Channel 2/Status/Status of input A
//     ExpEncB/输入/In/nState2 @bit 1 <-> ENC Status Channel 2/Status/Status of input B
//     ExpEncB/输入/In/nState2 @bit 2 <-> ENC Status Channel 2/Status/Status of input C
//     ExpEncB/输入/In/nState2 @bit 3 <-> ENC Status Channel 2/Status/Status of input gate
//     ExpEncB/输入/In/nState2 @bit 5 <-> ENC Status Channel 2/Status/TxPDO State
//     ExpEncB/输入/In/nState3 @bit 4 <-> ENC Status Channel 2/Status/Counter value out of range
//     ExpEncB/输入/In/nState3 @bit 2 <-> ENC Status Channel 2/Status/Direction inversion detected
//     ExpEncB/输入/In/nState3 @bit 1 <-> ENC Status Channel 2/Status/Latch extern 2 valid
//     ExpEncB/输入/In/nState3 <-> ENC Status Channel 2/Status/Software gate valid
//     ExpEncB/输入/In/nState3 @bit 3 <-> ENC Status Channel 2/Status/Status of extern latch
//     ExpEncB/输入/In/nState4 @bit 1 <-> WcState/InputToggle
//     ExpEncB/输入/In/nState4 <-> WcState/WcState
//     ExpEncB/输出/Out/nCtrl1 <-> ENC Control Channel 2/Control/Enable latch C
//     ExpEncB/输出/Out/nCtrl1 @bit 3 <-> ENC Control Channel 2/Control/Enable latch extern on negative edge
//     ExpEncB/输出/Out/nCtrl1 @bit 1 <-> ENC Control Channel 2/Control/Enable latch extern on positive edge
//     ExpEncB/输出/Out/nCtrl1 @bit 2 <-> ENC Control Channel 2/Control/Set counter
//     ExpEncB/输出/Out/nCtrl1 @bit 7 <-> ENC Control Channel 2/Control/Set counter on latch C
//     ExpEncB/输出/Out/nCtrl2 @bit 4 <-> ENC Control Channel 2/Control/Enable latch extern 2 on negative edge
//     ExpEncB/输出/Out/nCtrl2 @bit 3 <-> ENC Control Channel 2/Control/Enable latch extern 2 on positive edge
//     ExpEncB/输出/Out/nCtrl2 @bit 2 <-> ENC Control Channel 2/Control/Set counter on latch extern on negative edge
//     ExpEncB/输出/Out/nCtrl2 @bit 1 <-> ENC Control Channel 2/Control/Set counter on latch extern on positive edge
//     ExpEncB/输出/Out/nCtrl2 <-> ENC Control Channel 2/Control/Set software gate
//     ExpEncB/输出/Out/nDataOut1 <-> ENC Control Channel 2/Set counter value
//   NC-Task 1 SAF/Axes/FX1 <-> Device 2 (EtherCAT)/Box 1 (AMAX-4870)/Box 2 (AMAX-4870)/Box 3 (AMAX-4870)/Box 5 (SI6/SC6 2Ax)
//     Drive/Inputs/In/nDataIn1 <-> Module 1 (CiA)/Axis A to Master/1.A632 Following error actual value
//     Drive/Inputs/In/nDataIn3[0] <-> Module 1 (CiA)/Axis A to Master/1.A564 Torque actual value
//     Drive/Inputs/In/nDcOutputTime <-> InfoData/DcOutputShift
//     Drive/Inputs/In/nState1 <-> Module 1 (CiA)/Axis A to Master/1.A516 Statusword
//     Drive/Inputs/In/nState2 <-> Module 1 (CiA)/Axis A to Master/1.A516 Statusword @bit 8
//     Drive/Inputs/In/nState4 @bit 1 <-> WcState/InputToggle
//     Drive/Inputs/In/nState4 <-> WcState/WcState
//     Drive/Inputs/In/nState5 <-> Module 1 (CiA)/Axis A to Master/1.A542 Modes of operation display
//     Drive/Outputs/Out/nCtrl1 <-> Module 1 (CiA)/Axis A to Slave/1.A515 Controlword
//     Drive/Outputs/Out/nCtrl2 <-> Module 1 (CiA)/Axis A to Slave/1.A515 Controlword @bit 8
//     Drive/Outputs/Out/nCtrl5 <-> Module 1 (CiA)/Axis A to Slave/1.A541 Modes of operation
//     Drive/Outputs/Out/nDataOut1 <-> Module 1 (CiA)/Axis A to Slave/1.A567 Target position
//     Drive/Outputs/Out/nDataOut2 <-> Module 1 (CiA)/Axis A to Slave/1.A638 Target velocity
//     Drive/Outputs/Out/nDataOut3[0] <-> Module 1 (CiA)/Axis A to Slave/1.A593 Torque offset
//     Drive/Outputs/Out/nDataOut4[0] <-> Module 1 (CiA)/Axis A to Slave/1.A558 Target torque
//     Enc/Inputs/In/nDataIn1 <-> Module 1 (CiA)/Axis A to Master/1.A545 Position actual value
//     Enc/Inputs/In/nDataIn7 <-> Module 1 (CiA)/Axis A to Master/1.A553 Velocity actual value
//     Enc/Inputs/In/nDcInputTime <-> InfoData/DcInputShift
//     Enc/Inputs/In/nState4 @bit 1 <-> WcState/InputToggle
//     Enc/Inputs/In/nState4 <-> WcState/WcState
//   NC-Task 1 SAF/Axes/FX2 <-> Device 2 (EtherCAT)/Box 1 (AMAX-4870)/Box 2 (AMAX-4870)/Box 3 (AMAX-4870)/Box 5 (SI6/SC6 2Ax)
//     Drive/Inputs/In/nDataIn1 <-> Module 2 (CiA)/Axis B to Master/2.A632 Following error actual value
//     Drive/Inputs/In/nDataIn3[0] <-> Module 2 (CiA)/Axis B to Master/2.A564 Torque actual value
//     Drive/Inputs/In/nDcOutputTime <-> InfoData/DcOutputShift
//     Drive/Inputs/In/nState1 <-> Module 2 (CiA)/Axis B to Master/2.A516 Statusword
//     Drive/Inputs/In/nState2 <-> Module 2 (CiA)/Axis B to Master/2.A516 Statusword @bit 8
//     Drive/Inputs/In/nState4 @bit 1 <-> WcState/InputToggle
//     Drive/Inputs/In/nState4 <-> WcState/WcState
//     Drive/Inputs/In/nState5 <-> Module 2 (CiA)/Axis B to Master/2.A542 Modes of operation display
//     Drive/Outputs/Out/nCtrl1 <-> Module 2 (CiA)/Axis B to Slave/2.A515 Controlword
//     Drive/Outputs/Out/nCtrl2 <-> Module 2 (CiA)/Axis B to Slave/2.A515 Controlword @bit 8
//     Drive/Outputs/Out/nCtrl5 <-> Module 2 (CiA)/Axis B to Slave/2.A541 Modes of operation
//     Drive/Outputs/Out/nDataOut1 <-> Module 2 (CiA)/Axis B to Slave/2.A567 Target position
//     Drive/Outputs/Out/nDataOut2 <-> Module 2 (CiA)/Axis B to Slave/2.A638 Target velocity
//     Drive/Outputs/Out/nDataOut3[0] <-> Module 2 (CiA)/Axis B to Slave/2.A593 Torque offset
//     Drive/Outputs/Out/nDataOut4[0] <-> Module 2 (CiA)/Axis B to Slave/2.A558 Target torque
//     Enc/Inputs/In/nDataIn1 <-> Module 2 (CiA)/Axis B to Master/2.A545 Position actual value
//     Enc/Inputs/In/nDataIn7 <-> Module 2 (CiA)/Axis B to Master/2.A553 Velocity actual value
//     Enc/Inputs/In/nDcInputTime <-> InfoData/DcInputShift
//     Enc/Inputs/In/nState4 @bit 1 <-> WcState/InputToggle
//     Enc/Inputs/In/nState4 <-> WcState/WcState
//   NC-Task 1 SAF/Axes/MPG <-> Device 2 (EtherCAT)/Box 1 (AMAX-4870)/Box 2 (AMAX-4870)/Box 3 (AMAX-4870)/Box 4 (AMAX-4870)/Term 26 (EK1100)/Term 29 (EL5102)
//     Enc/Inputs/In/nDataIn1 <-> ENC Status Channel 1/Counter value
//     Enc/Inputs/In/nDataIn2 <-> ENC Status Channel 1/Latch value
//     Enc/Inputs/In/nState1 @bit 4 <-> ENC Status Channel 1/Status/Counter overflow
//     Enc/Inputs/In/nState1 @bit 3 <-> ENC Status Channel 1/Status/Counter underflow
//     Enc/Inputs/In/nState1 @bit 7 <-> ENC Status Channel 1/Status/Extrapolation stall
//     Enc/Inputs/In/nState1 <-> ENC Status Channel 1/Status/Latch C valid
//     Enc/Inputs/In/nState1 @bit 1 <-> ENC Status Channel 1/Status/Latch extern valid
//     Enc/Inputs/In/nState1 @bit 6 <-> ENC Status Channel 1/Status/Open circuit
//     Enc/Inputs/In/nState1 @bit 2 <-> ENC Status Channel 1/Status/Set counter done
//     Enc/Inputs/In/nState1 @bit 5 <-> ENC Status Channel 1/Status/Status of input status
//     Enc/Inputs/In/nState2 @bit 4 <-> ENC Status Channel 1/Status/Diag
//     Enc/Inputs/In/nState2 @bit 6 <-> ENC Status Channel 1/Status/Input cycle counter
//     Enc/Inputs/In/nState2 <-> ENC Status Channel 1/Status/Status of input A
//     Enc/Inputs/In/nState2 @bit 1 <-> ENC Status Channel 1/Status/Status of input B
//     Enc/Inputs/In/nState2 @bit 2 <-> ENC Status Channel 1/Status/Status of input C
//     Enc/Inputs/In/nState2 @bit 3 <-> ENC Status Channel 1/Status/Status of input gate
//     Enc/Inputs/In/nState2 @bit 5 <-> ENC Status Channel 1/Status/TxPDO State
//     Enc/Inputs/In/nState3 @bit 4 <-> ENC Status Channel 1/Status/Counter value out of range
//     Enc/Inputs/In/nState3 @bit 2 <-> ENC Status Channel 1/Status/Direction inversion detected
//     Enc/Inputs/In/nState3 @bit 1 <-> ENC Status Channel 1/Status/Latch extern 2 valid
//     Enc/Inputs/In/nState3 <-> ENC Status Channel 1/Status/Software gate valid
//     Enc/Inputs/In/nState3 @bit 3 <-> ENC Status Channel 1/Status/Status of extern latch
//     Enc/Inputs/In/nState4 @bit 1 <-> WcState/InputToggle
//     Enc/Inputs/In/nState4 <-> WcState/WcState
//     Enc/Outputs/Out/nCtrl1 <-> ENC Control Channel 1/Control/Enable latch C
//     Enc/Outputs/Out/nCtrl1 @bit 3 <-> ENC Control Channel 1/Control/Enable latch extern on negative edge
//     Enc/Outputs/Out/nCtrl1 @bit 1 <-> ENC Control Channel 1/Control/Enable latch extern on positive edge
//     Enc/Outputs/Out/nCtrl1 @bit 2 <-> ENC Control Channel 1/Control/Set counter
//     Enc/Outputs/Out/nCtrl1 @bit 7 <-> ENC Control Channel 1/Control/Set counter on latch C
//     Enc/Outputs/Out/nCtrl2 @bit 4 <-> ENC Control Channel 1/Control/Enable latch extern 2 on negative edge
//     Enc/Outputs/Out/nCtrl2 @bit 3 <-> ENC Control Channel 1/Control/Enable latch extern 2 on positive edge
//     Enc/Outputs/Out/nCtrl2 @bit 2 <-> ENC Control Channel 1/Control/Set counter on latch extern on negative edge
//     Enc/Outputs/Out/nCtrl2 @bit 1 <-> ENC Control Channel 1/Control/Set counter on latch extern on positive edge
//     Enc/Outputs/Out/nCtrl2 <-> ENC Control Channel 1/Control/Set software gate
//     Enc/Outputs/Out/nDataOut1 <-> ENC Control Channel 1/Set counter value
//   NC-Task 1 SAF/Axes/轴 19 <-> Device 2 (EtherCAT)/Box 1 (AMAX-4870)/驱动器 71 (CL3-E57H)
//     Drive/输入/In/nDataIn1 <-> TxPDO 1/Follow Error Actual Value
//     Drive/输入/In/nDcOutputTime <-> InfoData/DcOutputShift
//     Drive/输入/In/nState1 <-> TxPDO 1/StatusWord
//     Drive/输入/In/nState2 <-> TxPDO 1/StatusWord @bit 8
//     Drive/输入/In/nState4 @bit 1 <-> WcState/InputToggle
//     Drive/输入/In/nState4 <-> WcState/WcState
//     Drive/输入/In/nState5 <-> TxPDO 1/Modes of operation display
//     Drive/输出/Out/nCtrl1 <-> RxPDO 1/ControlWord
//     Drive/输出/Out/nCtrl2 <-> RxPDO 1/ControlWord @bit 8
//     Drive/输出/Out/nCtrl5 <-> RxPDO 1/Modes of operation
//     Drive/输出/Out/nDataOut1 <-> RxPDO 1/Target position
//     Drive/输出/Out/nDataOut2 <-> RxPDO 1/Target Velocity
//     Enc/输入/In/nDataIn1 <-> TxPDO 1/Position actual value
//     Enc/输入/In/nDataIn7 <-> TxPDO 1/Velocity actual value
//     Enc/输入/In/nDcInputTime <-> InfoData/DcInputShift
//     Enc/输入/In/nState4 @bit 1 <-> WcState/InputToggle
//     Enc/输入/In/nState4 <-> WcState/WcState
//   Main Instance <-> Device 1 (EtherCAT)
//     PlcTask Inputs/GetEtherSta.sNetId1 <-> InfoData/AmsNetId
//   Main Instance <-> Device 2 (EtherCAT)
//     PlcTask Inputs/GetEtherSta.sNetId2 <-> InfoData/AmsNetId
//   Main Instance <-> Device 2 (EtherCAT)/Box 1 (AMAX-4870)/Box 2 (AMAX-4870)/Box 14 (54632)
//     PlcTask Inputs/Sensor.sensorA.in_RawData[{0..3}] <-> Module 1 (IOL_4/4_I/O-Bytes)/TxPDO/input byte {0..3}  (4 links)
//     PlcTask Inputs/Sensor.sensorB.in_RawData[{0..3}] <-> Module 2 (IOL_4/4_I/O-Bytes)/TxPDO/input byte {0..3}  (4 links)
//     PlcTask Inputs/Sensor.sensorC.in_RawData[{0..3}] <-> Module 3 (IOL_4/4_I/O-Bytes)/TxPDO/input byte {0..3}  (4 links)
//     PlcTask Inputs/Sensor.sensorD.in_RawData[{0..3}] <-> Module 4 (IOL_4/4_I/O-Bytes)/TxPDO/input byte {0..3}  (4 links)
//     PlcTask Outputs/Sensor.sensorA.out_rawdata <-> Module 1 (IOL_4/4_I/O-Bytes)/RxPDO/output byte 0
//     PlcTask Outputs/Sensor.sensorB.out_rawdata <-> Module 2 (IOL_4/4_I/O-Bytes)/RxPDO/output byte 0
//     PlcTask Outputs/Sensor.sensorC.out_rawdata <-> Module 3 (IOL_4/4_I/O-Bytes)/RxPDO/output byte 0
//     PlcTask Outputs/Sensor.sensorD.out_rawdata <-> Module 4 (IOL_4/4_I/O-Bytes)/RxPDO/output byte 0
//   Main Instance <-> Device 2 (EtherCAT)/Box 1 (AMAX-4870)/Box 2 (AMAX-4870)/Box 3 (AMAX-4870)/Box 4 (AMAX-4870)/Term 26 (EK1100)/Term 28 (EL5102)
//     PlcTask Inputs/Axis.Encoder_FxA_Clamp.MDP5001_511_Input/MDP5001_511_Counter_value <-> ENC Status Channel 1/Counter value
//     PlcTask Inputs/Axis.Encoder_FxA_Clamp.MDP5001_511_Input/MDP5001_511_Latch_value <-> ENC Status Channel 1/Latch value
//     PlcTask Inputs/Axis.Encoder_FxA_Clamp.MDP5001_511_Input/MDP5001_511_Latch_value_2 <-> ENC Status Channel 1/Latch value 2
//     PlcTask Inputs/Axis.Encoder_FxA_Clamp.MDP5001_511_Input/MDP5001_511_Status <-> ENC Status Channel 1/Status
//     PlcTask Inputs/Axis.Encoder_FxB_Clamp.MDP5001_511_Input/MDP5001_511_Counter_value <-> ENC Status Channel 2/Counter value
//     PlcTask Inputs/Axis.Encoder_FxB_Clamp.MDP5001_511_Input/MDP5001_511_Latch_value <-> ENC Status Channel 2/Latch value
//     PlcTask Inputs/Axis.Encoder_FxB_Clamp.MDP5001_511_Input/MDP5001_511_Latch_value_2 <-> ENC Status Channel 2/Latch value 2
//     PlcTask Inputs/Axis.Encoder_FxB_Clamp.MDP5001_511_Input/MDP5001_511_Status <-> ENC Status Channel 2/Status
//     PlcTask Outputs/Axis.Encoder_FxA_Clamp.MDP5001_511_Output/MDP5001_511_Control <-> ENC Control Channel 1/Control
//     PlcTask Outputs/Axis.Encoder_FxA_Clamp.MDP5001_511_Output/MDP5001_511_Set_counter_value <-> ENC Control Channel 1/Set counter value
//     PlcTask Outputs/Axis.Encoder_FxB_Clamp.MDP5001_511_Output/MDP5001_511_Control <-> ENC Control Channel 2/Control
//     PlcTask Outputs/Axis.Encoder_FxB_Clamp.MDP5001_511_Output/MDP5001_511_Set_counter_value <-> ENC Control Channel 2/Set counter value
//   Main Instance <-> Device 2 (EtherCAT)/Box 1 (AMAX-4870)/Box 2 (AMAX-4870)/Box 3 (AMAX-4870)/Box 4 (AMAX-4870)/Term 26 (EK1100)/Term 30 (EL5102)
//     PlcTask Inputs/Axis.Encoder_FxA_ExPosEnc.MDP5001_511_Input/MDP5001_511_Counter_value <-> ENC Status Channel 1/Counter value
//     PlcTask Inputs/Axis.Encoder_FxA_ExPosEnc.MDP5001_511_Input/MDP5001_511_Latch_value <-> ENC Status Channel 1/Latch value
//     PlcTask Inputs/Axis.Encoder_FxA_ExPosEnc.MDP5001_511_Input/MDP5001_511_Latch_value_2 <-> ENC Status Channel 1/Latch value 2
//     PlcTask Inputs/Axis.Encoder_FxA_ExPosEnc.MDP5001_511_Input/MDP5001_511_Status <-> ENC Status Channel 1/Status
//     PlcTask Inputs/Axis.Encoder_FxB_ExPosEnc.MDP5001_511_Input/MDP5001_511_Counter_value <-> ENC Status Channel 2/Counter value
//     PlcTask Inputs/Axis.Encoder_FxB_ExPosEnc.MDP5001_511_Input/MDP5001_511_Latch_value <-> ENC Status Channel 2/Latch value
//     PlcTask Inputs/Axis.Encoder_FxB_ExPosEnc.MDP5001_511_Input/MDP5001_511_Latch_value_2 <-> ENC Status Channel 2/Latch value 2
//     PlcTask Inputs/Axis.Encoder_FxB_ExPosEnc.MDP5001_511_Input/MDP5001_511_Status <-> ENC Status Channel 2/Status
//     PlcTask Outputs/Axis.Encoder_FxA_ExPosEnc.MDP5001_511_Output/MDP5001_511_Control <-> ENC Control Channel 1/Control
//     PlcTask Outputs/Axis.Encoder_FxA_ExPosEnc.MDP5001_511_Output/MDP5001_511_Set_counter_value <-> ENC Control Channel 1/Set counter value
//     PlcTask Outputs/Axis.Encoder_FxB_ExPosEnc.MDP5001_511_Output/MDP5001_511_Control <-> ENC Control Channel 2/Control
//     PlcTask Outputs/Axis.Encoder_FxB_ExPosEnc.MDP5001_511_Output/MDP5001_511_Set_counter_value <-> ENC Control Channel 2/Set counter value
//   Main Instance <-> NC-Task 1 SAF/Axes/AX
//     PlcTask Inputs/Axis.Axis_AX.NcToPlc <-> Outputs/ToPlc
//     PlcTask Outputs/Axis.Axis_AX.PlcToNc <-> Inputs/FromPlc
//   Main Instance <-> NC-Task 1 SAF/Axes/AY
//     PlcTask Inputs/Axis.Axis_AY.NcToPlc <-> Outputs/ToPlc
//     PlcTask Outputs/Axis.Axis_AY.PlcToNc <-> Inputs/FromPlc
//   Main Instance <-> NC-Task 1 SAF/Axes/AZ1
//     PlcTask Inputs/Axis.Axis_AZ1.NcToPlc <-> Outputs/ToPlc
//     PlcTask Outputs/Axis.Axis_AZ1.PlcToNc <-> Inputs/FromPlc
//   Main Instance <-> NC-Task 1 SAF/Axes/AZ2
//     PlcTask Inputs/Axis.Axis_AZ2.NcToPlc <-> Outputs/ToPlc
//     PlcTask Outputs/Axis.Axis_AZ2.PlcToNc <-> Inputs/FromPlc
//   Main Instance <-> NC-Task 1 SAF/Axes/BX
//     PlcTask Inputs/Axis.Axis_BX.NcToPlc <-> Outputs/ToPlc
//     PlcTask Outputs/Axis.Axis_BX.PlcToNc <-> Inputs/FromPlc
//   Main Instance <-> NC-Task 1 SAF/Axes/BY1
//     PlcTask Inputs/Axis.Axis_BY1.NcToPlc <-> Outputs/ToPlc
//     PlcTask Outputs/Axis.Axis_BY1.PlcToNc <-> Inputs/FromPlc
//   Main Instance <-> NC-Task 1 SAF/Axes/BY2
//     PlcTask Inputs/Axis.Axis_BY2.NcToPlc <-> Outputs/ToPlc
//     PlcTask Outputs/Axis.Axis_BY2.PlcToNc <-> Inputs/FromPlc
//   Main Instance <-> NC-Task 1 SAF/Axes/BZ
//     PlcTask Inputs/Axis.Axis_BZ.NcToPlc <-> Outputs/ToPlc
//     PlcTask Outputs/Axis.Axis_BZ.PlcToNc <-> Inputs/FromPlc
//   Main Instance <-> NC-Task 1 SAF/Axes/CX
//     PlcTask Inputs/Axis.Axis_CX.NcToPlc <-> Outputs/ToPlc
//     PlcTask Outputs/Axis.Axis_CX.PlcToNc <-> Inputs/FromPlc
//   Main Instance <-> NC-Task 1 SAF/Axes/CY
//     PlcTask Inputs/Axis.Axis_CY.NcToPlc <-> Outputs/ToPlc
//     PlcTask Outputs/Axis.Axis_CY.PlcToNc <-> Inputs/FromPlc
//   Main Instance <-> NC-Task 1 SAF/Axes/CZ1
//     PlcTask Inputs/Axis.Axis_CZ1.NcToPlc <-> Outputs/ToPlc
//     PlcTask Outputs/Axis.Axis_CZ1.PlcToNc <-> Inputs/FromPlc
//   Main Instance <-> NC-Task 1 SAF/Axes/CZ2
//     PlcTask Inputs/Axis.Axis_CZ2.NcToPlc <-> Outputs/ToPlc
//     PlcTask Outputs/Axis.Axis_CZ2.PlcToNc <-> Inputs/FromPlc
//   Main Instance <-> NC-Task 1 SAF/Axes/DX
//     PlcTask Inputs/Axis.Axis_DX.NcToPlc <-> Outputs/ToPlc
//     PlcTask Outputs/Axis.Axis_DX.PlcToNc <-> Inputs/FromPlc
//   Main Instance <-> NC-Task 1 SAF/Axes/DY
//     PlcTask Inputs/Axis.Axis_DY.NcToPlc <-> Outputs/ToPlc
//     PlcTask Outputs/Axis.Axis_DY.PlcToNc <-> Inputs/FromPlc
//   Main Instance <-> NC-Task 1 SAF/Axes/DZ
//     PlcTask Inputs/Axis.Axis_DZ.NcToPlc <-> Outputs/ToPlc
//     PlcTask Outputs/Axis.Axis_DZ.PlcToNc <-> Inputs/FromPlc
//   Main Instance <-> NC-Task 1 SAF/Axes/FX1
//     PlcTask Inputs/Axis.Axis_FX1.NcToPlc <-> Outputs/ToPlc
//     PlcTask Outputs/Axis.Axis_FX1.PlcToNc <-> Inputs/FromPlc
//   Main Instance <-> NC-Task 1 SAF/Axes/FX2
//     PlcTask Inputs/Axis.Axis_FX2.NcToPlc <-> Outputs/ToPlc
//     PlcTask Outputs/Axis.Axis_FX2.PlcToNc <-> Inputs/FromPlc
//   Main Instance <-> NC-Task 1 SAF/Axes/MPG
//     PlcTask Inputs/Jog_MPG.AxisMPG.NcToPlc <-> Outputs/ToPlc
//     PlcTask Outputs/Jog_MPG.AxisMPG.PlcToNc <-> Inputs/FromPlc
//   IO_Main_Task Instance <-> Device 1 (EtherCAT)/Term 1 (EK1200)/Term 10 (EL2409)
//     IO_Task Inputs/EtherCAT.MainMod_9.State <-> InfoData/State
//     IO_Task Inputs/EtherCAT.MainMod_9.WcState <-> WcState/WcState
//     IO_Task Outputs/EtherCAT.MainMod_9.Output[{1..16}] <-> Channel {1..16}/Output  (16 links)
//   IO_Main_Task Instance <-> Device 1 (EtherCAT)/Term 1 (EK1200)/Term 2 (EL1409)
//     IO_Task Inputs/EtherCAT.MainMod_1.InputToggle <-> WcState/InputToggle
//     IO_Task Inputs/EtherCAT.MainMod_1.Input[{1..16}] <-> DIP Inputs/Input Channel {1..16}  (16 links)
//     IO_Task Inputs/EtherCAT.MainMod_1.State <-> InfoData/State
//     IO_Task Inputs/EtherCAT.MainMod_1.WcState <-> WcState/WcState
//   IO_Main_Task Instance <-> Device 1 (EtherCAT)/Term 1 (EK1200)/Term 3 (EL1409)
//     IO_Task Inputs/EtherCAT.MainMod_2.InputToggle <-> WcState/InputToggle
//     IO_Task Inputs/EtherCAT.MainMod_2.Input[{1..16}] <-> DIP Inputs/Input Channel {1..16}  (16 links)
//     IO_Task Inputs/EtherCAT.MainMod_2.State <-> InfoData/State
//     IO_Task Inputs/EtherCAT.MainMod_2.WcState <-> WcState/WcState
//   IO_Main_Task Instance <-> Device 1 (EtherCAT)/Term 1 (EK1200)/Term 4 (EL1409)
//     IO_Task Inputs/EtherCAT.MainMod_3.InputToggle <-> WcState/InputToggle
//     IO_Task Inputs/EtherCAT.MainMod_3.Input[{1..16}] <-> DIP Inputs/Input Channel {1..16}  (16 links)
//     IO_Task Inputs/EtherCAT.MainMod_3.State <-> InfoData/State
//     IO_Task Inputs/EtherCAT.MainMod_3.WcState <-> WcState/WcState
//   IO_Main_Task Instance <-> Device 1 (EtherCAT)/Term 1 (EK1200)/Term 5 (EL1409)
//     IO_Task Inputs/EtherCAT.MainMod_4.InputToggle <-> WcState/InputToggle
//     IO_Task Inputs/EtherCAT.MainMod_4.Input[{1..16}] <-> DIP Inputs/Input Channel {1..16}  (16 links)
//     IO_Task Inputs/EtherCAT.MainMod_4.State <-> InfoData/State
//     IO_Task Inputs/EtherCAT.MainMod_4.WcState <-> WcState/WcState
//   IO_Main_Task Instance <-> Device 1 (EtherCAT)/Term 1 (EK1200)/Term 6 (EL1409)
//     IO_Task Inputs/EtherCAT.MainMod_5.InputToggle <-> WcState/InputToggle
//     IO_Task Inputs/EtherCAT.MainMod_5.Input[{1..16}] <-> DIP Inputs/Input Channel {1..16}  (16 links)
//     IO_Task Inputs/EtherCAT.MainMod_5.State <-> InfoData/State
//     IO_Task Inputs/EtherCAT.MainMod_5.WcState <-> WcState/WcState
//   IO_Main_Task Instance <-> Device 1 (EtherCAT)/Term 1 (EK1200)/Term 7 (EL1409)
//     IO_Task Inputs/EtherCAT.MainMod_6.InputToggle <-> WcState/InputToggle
//     IO_Task Inputs/EtherCAT.MainMod_6.Input[{1..16}] <-> DIP Inputs/Input Channel {1..16}  (16 links)
//     IO_Task Inputs/EtherCAT.MainMod_6.State <-> InfoData/State
//     IO_Task Inputs/EtherCAT.MainMod_6.WcState <-> WcState/WcState
//   IO_Main_Task Instance <-> Device 1 (EtherCAT)/Term 1 (EK1200)/Term 8 (EL2409)
//     IO_Task Inputs/EtherCAT.MainMod_7.State <-> InfoData/State
//     IO_Task Inputs/EtherCAT.MainMod_7.WcState <-> WcState/WcState
//     IO_Task Outputs/EtherCAT.MainMod_7.Output[{1..16}] <-> Channel {1..16}/Output  (16 links)
//   IO_Main_Task Instance <-> Device 1 (EtherCAT)/Term 1 (EK1200)/Term 9 (EL2409)
//     IO_Task Inputs/EtherCAT.MainMod_8.State <-> InfoData/State
//     IO_Task Inputs/EtherCAT.MainMod_8.WcState <-> WcState/WcState
//     IO_Task Outputs/EtherCAT.MainMod_8.Output[{1..16}] <-> Channel {1..16}/Output  (16 links)
//   IO_Main_Task Instance <-> Device 2 (EtherCAT)/Box 1 (AMAX-4870)/Box 2 (AMAX-4870)/Box 14 (54632)
//     IO_Task Inputs/EtherCAT.Murr_Mod.Input <-> TxPDO Mapping of Digital Inputs/PD (I/Q Pin2 + C/Q Pin4)
//     IO_Task Inputs/EtherCAT.Murr_Mod.InputToggle <-> WcState/InputToggle
//     IO_Task Inputs/EtherCAT.Murr_Mod.Io_State[{0..7}] <-> TxPDO Mapping of Status Data/State of IO-Link Port X{0..7}  (8 links)
//     IO_Task Inputs/EtherCAT.Murr_Mod.State <-> InfoData/State
//     IO_Task Inputs/EtherCAT.Murr_Mod.WcState <-> WcState/WcState
//   IO_Main_Task Instance <-> Main/Main Instance
//     IO_Task Inputs/MainIO.IO107.Out[10] <-> PlcTask Outputs/IO.q110
//     IO_Task Inputs/MainIO.IO107.Out[11] <-> PlcTask Outputs/IO.q111
//     IO_Task Inputs/MainIO.IO107.Out[12] <-> PlcTask Outputs/IO.q112
//     IO_Task Inputs/MainIO.IO107.Out[13] <-> PlcTask Outputs/IO.q113
//     IO_Task Inputs/MainIO.IO107.Out[14] <-> PlcTask Outputs/IO.q114
//     IO_Task Inputs/MainIO.IO107.Out[15] <-> PlcTask Outputs/IO.q115
//     IO_Task Inputs/MainIO.IO107.Out[16] <-> PlcTask Outputs/IO.q116
//     IO_Task Inputs/MainIO.IO107.Out[1] <-> PlcTask Outputs/IO.q101
//     IO_Task Inputs/MainIO.IO107.Out[2] <-> PlcTask Outputs/IO.q102
//     IO_Task Inputs/MainIO.IO107.Out[3] <-> PlcTask Outputs/IO.q103
//     IO_Task Inputs/MainIO.IO107.Out[4] <-> PlcTask Outputs/IO.q104
//     IO_Task Inputs/MainIO.IO107.Out[5] <-> PlcTask Outputs/IO.q105
//     IO_Task Inputs/MainIO.IO107.Out[6] <-> PlcTask Outputs/IO.q106
//     IO_Task Inputs/MainIO.IO107.Out[7] <-> PlcTask Outputs/IO.q107
//     IO_Task Inputs/MainIO.IO107.Out[8] <-> PlcTask Outputs/IO.q108
//     IO_Task Inputs/MainIO.IO107.Out[9] <-> PlcTask Outputs/IO.q109
//     IO_Task Inputs/MainIO.IO108.Out[10] <-> PlcTask Outputs/IO.q210
//     IO_Task Inputs/MainIO.IO108.Out[11] <-> PlcTask Outputs/IO.q211
//     IO_Task Inputs/MainIO.IO108.Out[12] <-> PlcTask Outputs/IO.q212
//     IO_Task Inputs/MainIO.IO108.Out[13] <-> PlcTask Outputs/IO.q213
//     IO_Task Inputs/MainIO.IO108.Out[14] <-> PlcTask Outputs/IO.q214
//     IO_Task Inputs/MainIO.IO108.Out[15] <-> PlcTask Outputs/IO.q215
//     IO_Task Inputs/MainIO.IO108.Out[16] <-> PlcTask Outputs/IO.q216
//     IO_Task Inputs/MainIO.IO108.Out[1] <-> PlcTask Outputs/IO.q201
//     IO_Task Inputs/MainIO.IO108.Out[2] <-> PlcTask Outputs/IO.q202
//     IO_Task Inputs/MainIO.IO108.Out[3] <-> PlcTask Outputs/IO.q203
//     IO_Task Inputs/MainIO.IO108.Out[4] <-> PlcTask Outputs/IO.q204
//     IO_Task Inputs/MainIO.IO108.Out[5] <-> PlcTask Outputs/IO.q205
//     IO_Task Inputs/MainIO.IO108.Out[6] <-> PlcTask Outputs/IO.q206
//     IO_Task Inputs/MainIO.IO108.Out[7] <-> PlcTask Outputs/IO.q207
//     IO_Task Inputs/MainIO.IO108.Out[8] <-> PlcTask Outputs/IO.q208
//     IO_Task Inputs/MainIO.IO108.Out[9] <-> PlcTask Outputs/IO.q209
//     IO_Task Inputs/MainIO.IO109.Out[10] <-> PlcTask Outputs/IO.q310
//     IO_Task Inputs/MainIO.IO109.Out[11] <-> PlcTask Outputs/IO.q311
//     IO_Task Inputs/MainIO.IO109.Out[12] <-> PlcTask Outputs/IO.q312
//     IO_Task Inputs/MainIO.IO109.Out[13] <-> PlcTask Outputs/IO.q313
//     IO_Task Inputs/MainIO.IO109.Out[14] <-> PlcTask Outputs/IO.q314
//     IO_Task Inputs/MainIO.IO109.Out[15] <-> PlcTask Outputs/IO.q315
//     IO_Task Inputs/MainIO.IO109.Out[16] <-> PlcTask Outputs/IO.q316
//     IO_Task Inputs/MainIO.IO109.Out[1] <-> PlcTask Outputs/IO.q301
//     IO_Task Inputs/MainIO.IO109.Out[2] <-> PlcTask Outputs/IO.q302
//     IO_Task Inputs/MainIO.IO109.Out[3] <-> PlcTask Outputs/IO.q303
//     IO_Task Inputs/MainIO.IO109.Out[4] <-> PlcTask Outputs/IO.q304
//     IO_Task Inputs/MainIO.IO109.Out[5] <-> PlcTask Outputs/IO.q305
//     IO_Task Inputs/MainIO.IO109.Out[6] <-> PlcTask Outputs/IO.q306
//     IO_Task Inputs/MainIO.IO109.Out[7] <-> PlcTask Outputs/IO.q307
//     IO_Task Inputs/MainIO.IO109.Out[8] <-> PlcTask Outputs/IO.q308
//     IO_Task Inputs/MainIO.IO109.Out[9] <-> PlcTask Outputs/IO.q309
//     IO_Task Outputs/MainIO.IO101.In[10] <-> PlcTask Inputs/IO.i110
//     IO_Task Outputs/MainIO.IO101.In[11] <-> PlcTask Inputs/IO.i111
//     IO_Task Outputs/MainIO.IO101.In[12] <-> PlcTask Inputs/IO.i112
//     IO_Task Outputs/MainIO.IO101.In[13] <-> PlcTask Inputs/IO.i113
//     IO_Task Outputs/MainIO.IO101.In[14] <-> PlcTask Inputs/IO.i114
//     IO_Task Outputs/MainIO.IO101.In[15] <-> PlcTask Inputs/IO.i115
//     IO_Task Outputs/MainIO.IO101.In[16] <-> PlcTask Inputs/IO.i116
//     IO_Task Outputs/MainIO.IO101.In[1] <-> PlcTask Inputs/IO.i101
//     IO_Task Outputs/MainIO.IO101.In[2] <-> PlcTask Inputs/IO.i102
//     IO_Task Outputs/MainIO.IO101.In[3] <-> PlcTask Inputs/IO.i103
//     IO_Task Outputs/MainIO.IO101.In[4] <-> PlcTask Inputs/IO.i104
//     IO_Task Outputs/MainIO.IO101.In[5] <-> PlcTask Inputs/IO.i105
//     IO_Task Outputs/MainIO.IO101.In[6] <-> PlcTask Inputs/IO.i106
//     IO_Task Outputs/MainIO.IO101.In[7] <-> PlcTask Inputs/IO.i107
//     IO_Task Outputs/MainIO.IO101.In[8] <-> PlcTask Inputs/IO.i108
//     IO_Task Outputs/MainIO.IO101.In[9] <-> PlcTask Inputs/IO.i109
//     IO_Task Outputs/MainIO.IO102.In[10] <-> PlcTask Inputs/IO.i210
//     IO_Task Outputs/MainIO.IO102.In[11] <-> PlcTask Inputs/IO.i211
//     IO_Task Outputs/MainIO.IO102.In[12] <-> PlcTask Inputs/IO.i212
//     IO_Task Outputs/MainIO.IO102.In[13] <-> PlcTask Inputs/IO.i213
//     IO_Task Outputs/MainIO.IO102.In[14] <-> PlcTask Inputs/IO.i214
//     IO_Task Outputs/MainIO.IO102.In[15] <-> PlcTask Inputs/IO.i215
//     IO_Task Outputs/MainIO.IO102.In[16] <-> PlcTask Inputs/IO.i216
//     IO_Task Outputs/MainIO.IO102.In[1] <-> PlcTask Inputs/IO.i201
//     IO_Task Outputs/MainIO.IO102.In[2] <-> PlcTask Inputs/IO.i202
//     IO_Task Outputs/MainIO.IO102.In[3] <-> PlcTask Inputs/IO.i203
//     IO_Task Outputs/MainIO.IO102.In[4] <-> PlcTask Inputs/IO.i204
//     IO_Task Outputs/MainIO.IO102.In[5] <-> PlcTask Inputs/IO.i205
//     IO_Task Outputs/MainIO.IO102.In[6] <-> PlcTask Inputs/IO.i206
//     IO_Task Outputs/MainIO.IO102.In[7] <-> PlcTask Inputs/IO.i207
//     IO_Task Outputs/MainIO.IO102.In[8] <-> PlcTask Inputs/IO.i208
//     IO_Task Outputs/MainIO.IO102.In[9] <-> PlcTask Inputs/IO.i209
//     IO_Task Outputs/MainIO.IO103.In[10] <-> PlcTask Inputs/IO.i310
//     IO_Task Outputs/MainIO.IO103.In[11] <-> PlcTask Inputs/IO.i311
//     IO_Task Outputs/MainIO.IO103.In[12] <-> PlcTask Inputs/IO.i312
//     IO_Task Outputs/MainIO.IO103.In[13] <-> PlcTask Inputs/IO.i313
//     IO_Task Outputs/MainIO.IO103.In[14] <-> PlcTask Inputs/IO.i314
//     IO_Task Outputs/MainIO.IO103.In[15] <-> PlcTask Inputs/IO.i315
//     IO_Task Outputs/MainIO.IO103.In[16] <-> PlcTask Inputs/IO.i316
//     IO_Task Outputs/MainIO.IO103.In[1] <-> PlcTask Inputs/IO.i301
//     IO_Task Outputs/MainIO.IO103.In[2] <-> PlcTask Inputs/IO.i302
//     IO_Task Outputs/MainIO.IO103.In[3] <-> PlcTask Inputs/IO.i303
//     IO_Task Outputs/MainIO.IO103.In[4] <-> PlcTask Inputs/IO.i304
//     IO_Task Outputs/MainIO.IO103.In[5] <-> PlcTask Inputs/IO.i305
//     IO_Task Outputs/MainIO.IO103.In[6] <-> PlcTask Inputs/IO.i306
//     IO_Task Outputs/MainIO.IO103.In[7] <-> PlcTask Inputs/IO.i307
//     IO_Task Outputs/MainIO.IO103.In[8] <-> PlcTask Inputs/IO.i308
//     IO_Task Outputs/MainIO.IO103.In[9] <-> PlcTask Inputs/IO.i309
//     IO_Task Outputs/MainIO.IO104.In[10] <-> PlcTask Inputs/IO.i410
//     IO_Task Outputs/MainIO.IO104.In[11] <-> PlcTask Inputs/IO.i411
//     IO_Task Outputs/MainIO.IO104.In[12] <-> PlcTask Inputs/IO.i412
//     IO_Task Outputs/MainIO.IO104.In[13] <-> PlcTask Inputs/IO.i413
//     IO_Task Outputs/MainIO.IO104.In[14] <-> PlcTask Inputs/IO.i414
//     IO_Task Outputs/MainIO.IO104.In[15] <-> PlcTask Inputs/IO.i415
//     IO_Task Outputs/MainIO.IO104.In[16] <-> PlcTask Inputs/IO.i416
//     IO_Task Outputs/MainIO.IO104.In[1] <-> PlcTask Inputs/IO.i401
//     IO_Task Outputs/MainIO.IO104.In[2] <-> PlcTask Inputs/IO.i402
//     IO_Task Outputs/MainIO.IO104.In[3] <-> PlcTask Inputs/IO.i403
//     IO_Task Outputs/MainIO.IO104.In[4] <-> PlcTask Inputs/IO.i404
//     IO_Task Outputs/MainIO.IO104.In[5] <-> PlcTask Inputs/IO.i405
//     IO_Task Outputs/MainIO.IO104.In[6] <-> PlcTask Inputs/IO.i406
//     IO_Task Outputs/MainIO.IO104.In[7] <-> PlcTask Inputs/IO.i407
//     IO_Task Outputs/MainIO.IO104.In[8] <-> PlcTask Inputs/IO.i408
//     IO_Task Outputs/MainIO.IO104.In[9] <-> PlcTask Inputs/IO.i409
//     IO_Task Outputs/MainIO.IO105.In[10] <-> PlcTask Inputs/IO.i510
//     IO_Task Outputs/MainIO.IO105.In[11] <-> PlcTask Inputs/IO.i511
//     IO_Task Outputs/MainIO.IO105.In[12] <-> PlcTask Inputs/IO.i512
//     IO_Task Outputs/MainIO.IO105.In[13] <-> PlcTask Inputs/IO.i513
//     IO_Task Outputs/MainIO.IO105.In[14] <-> PlcTask Inputs/IO.i514
//     IO_Task Outputs/MainIO.IO105.In[15] <-> PlcTask Inputs/IO.i515
//     IO_Task Outputs/MainIO.IO105.In[16] <-> PlcTask Inputs/IO.i516
//     IO_Task Outputs/MainIO.IO105.In[1] <-> PlcTask Inputs/IO.i501
//     IO_Task Outputs/MainIO.IO105.In[2] <-> PlcTask Inputs/IO.i502
//     IO_Task Outputs/MainIO.IO105.In[3] <-> PlcTask Inputs/IO.i503
//     IO_Task Outputs/MainIO.IO105.In[4] <-> PlcTask Inputs/IO.i504
//     IO_Task Outputs/MainIO.IO105.In[5] <-> PlcTask Inputs/IO.i505
//     IO_Task Outputs/MainIO.IO105.In[6] <-> PlcTask Inputs/IO.i506
//     IO_Task Outputs/MainIO.IO105.In[7] <-> PlcTask Inputs/IO.i507
//     IO_Task Outputs/MainIO.IO105.In[8] <-> PlcTask Inputs/IO.i508
//     IO_Task Outputs/MainIO.IO105.In[9] <-> PlcTask Inputs/IO.i509
//     IO_Task Outputs/MainIO.IO106.In[10] <-> PlcTask Inputs/IO.i610
//     IO_Task Outputs/MainIO.IO106.In[11] <-> PlcTask Inputs/IO.i611
//     IO_Task Outputs/MainIO.IO106.In[12] <-> PlcTask Inputs/IO.i612
//     IO_Task Outputs/MainIO.IO106.In[13] <-> PlcTask Inputs/IO.i613
//     IO_Task Outputs/MainIO.IO106.In[14] <-> PlcTask Inputs/IO.i614
//     IO_Task Outputs/MainIO.IO106.In[15] <-> PlcTask Inputs/IO.i615
//     IO_Task Outputs/MainIO.IO106.In[16] <-> PlcTask Inputs/IO.i616
//     IO_Task Outputs/MainIO.IO106.In[1] <-> PlcTask Inputs/IO.i601
//     IO_Task Outputs/MainIO.IO106.In[2] <-> PlcTask Inputs/IO.i602
//     IO_Task Outputs/MainIO.IO106.In[3] <-> PlcTask Inputs/IO.i603
//     IO_Task Outputs/MainIO.IO106.In[4] <-> PlcTask Inputs/IO.i604
//     IO_Task Outputs/MainIO.IO106.In[5] <-> PlcTask Inputs/IO.i605
//     IO_Task Outputs/MainIO.IO106.In[6] <-> PlcTask Inputs/IO.i606
//     IO_Task Outputs/MainIO.IO106.In[7] <-> PlcTask Inputs/IO.i607
//     IO_Task Outputs/MainIO.IO106.In[8] <-> PlcTask Inputs/IO.i608
//     IO_Task Outputs/MainIO.IO106.In[9] <-> PlcTask Inputs/IO.i609
//     IO_Task Outputs/MainIO.IO401.In[10] <-> PlcTask Inputs/IO.i710
//     IO_Task Outputs/MainIO.IO401.In[11] <-> PlcTask Inputs/IO.i711
//     IO_Task Outputs/MainIO.IO401.In[12] <-> PlcTask Inputs/IO.i712
//     IO_Task Outputs/MainIO.IO401.In[13] <-> PlcTask Inputs/IO.i713
//     IO_Task Outputs/MainIO.IO401.In[14] <-> PlcTask Inputs/IO.i714
//     IO_Task Outputs/MainIO.IO401.In[15] <-> PlcTask Inputs/IO.i715
//     IO_Task Outputs/MainIO.IO401.In[16] <-> PlcTask Inputs/IO.i716
//     IO_Task Outputs/MainIO.IO401.In[1] <-> PlcTask Inputs/IO.i701
//     IO_Task Outputs/MainIO.IO401.In[2] <-> PlcTask Inputs/IO.i702
//     IO_Task Outputs/MainIO.IO401.In[3] <-> PlcTask Inputs/IO.i703
//     IO_Task Outputs/MainIO.IO401.In[4] <-> PlcTask Inputs/IO.i704
//     IO_Task Outputs/MainIO.IO401.In[5] <-> PlcTask Inputs/IO.i705
//     IO_Task Outputs/MainIO.IO401.In[6] <-> PlcTask Inputs/IO.i706
//     IO_Task Outputs/MainIO.IO401.In[7] <-> PlcTask Inputs/IO.i707
//     IO_Task Outputs/MainIO.IO401.In[8] <-> PlcTask Inputs/IO.i708
//     IO_Task Outputs/MainIO.IO401.In[9] <-> PlcTask Inputs/IO.i709
//   IO_External_Task Instance <-> Device 2 (EtherCAT)/Box 1 (AMAX-4870)/Box 51 (BL 570)/DI570 10 (DI 570)
//     Main_IO_Task Inputs/EtherCAT.LoadMod_3.InputToggle <-> WcState/InputToggle
//     Main_IO_Task Inputs/EtherCAT.LoadMod_3.Input[{1..16}] <-> DI Mapping/DI{0..15} Value  (16 links)
//     Main_IO_Task Inputs/EtherCAT.LoadMod_3.State <-> InfoData/State
//     Main_IO_Task Inputs/EtherCAT.LoadMod_3.WcState <-> WcState/WcState
//   IO_External_Task Instance <-> Device 2 (EtherCAT)/Box 1 (AMAX-4870)/Box 51 (BL 570)/DI570 11 (DI 570)
//     Main_IO_Task Inputs/EtherCAT.LoadMod_4.InputToggle <-> WcState/InputToggle
//     Main_IO_Task Inputs/EtherCAT.LoadMod_4.Input[{1..16}] <-> DI Mapping/DI{0..15} Value  (16 links)
//     Main_IO_Task Inputs/EtherCAT.LoadMod_4.State <-> InfoData/State
//     Main_IO_Task Inputs/EtherCAT.LoadMod_4.WcState <-> WcState/WcState
//   IO_External_Task Instance <-> Device 2 (EtherCAT)/Box 1 (AMAX-4870)/Box 51 (BL 570)/DI570 8 (DI 570)
//     Main_IO_Task Inputs/EtherCAT.LoadMod_1.InputToggle <-> WcState/InputToggle
//     Main_IO_Task Inputs/EtherCAT.LoadMod_1.Input[{1..16}] <-> DI Mapping/DI{0..15} Value  (16 links)
//     Main_IO_Task Inputs/EtherCAT.LoadMod_1.State <-> InfoData/State
//     Main_IO_Task Inputs/EtherCAT.LoadMod_1.WcState <-> WcState/WcState
//   IO_External_Task Instance <-> Device 2 (EtherCAT)/Box 1 (AMAX-4870)/Box 51 (BL 570)/DI570 9 (DI 570)
//     Main_IO_Task Inputs/EtherCAT.LoadMod_2.InputToggle <-> WcState/InputToggle
//     Main_IO_Task Inputs/EtherCAT.LoadMod_2.Input[{1..16}] <-> DI Mapping/DI{0..15} Value  (16 links)
//     Main_IO_Task Inputs/EtherCAT.LoadMod_2.State <-> InfoData/State
//     Main_IO_Task Inputs/EtherCAT.LoadMod_2.WcState <-> WcState/WcState
//   IO_External_Task Instance <-> Device 2 (EtherCAT)/Box 1 (AMAX-4870)/Box 51 (BL 570)/DO570 4 (DO 570)
//     Main_IO_Task Inputs/EtherCAT.LoadMod_5.Output_ShortCircuit[{1..16}] <-> DO SC State Mapping/DO{0..15} SC State  (16 links)
//     Main_IO_Task Inputs/EtherCAT.LoadMod_5.State <-> InfoData/State
//     Main_IO_Task Inputs/EtherCAT.LoadMod_5.WcState <-> WcState/WcState
//     Main_IO_Task Outputs/EtherCAT.LoadMod_5.Output[{1..16}] <-> DO Mapping/DO{0..15} Value  (16 links)
//   IO_External_Task Instance <-> Device 2 (EtherCAT)/Box 1 (AMAX-4870)/Box 51 (BL 570)/DO570 5 (DO 570)
//     Main_IO_Task Inputs/EtherCAT.LoadMod_6.Output_ShortCircuit[{1..16}] <-> DO SC State Mapping/DO{0..15} SC State  (16 links)
//     Main_IO_Task Inputs/EtherCAT.LoadMod_6.State <-> InfoData/State
//     Main_IO_Task Inputs/EtherCAT.LoadMod_6.WcState <-> WcState/WcState
//     Main_IO_Task Outputs/EtherCAT.LoadMod_6.Output[{1..16}] <-> DO Mapping/DO{0..15} Value  (16 links)
//   IO_External_Task Instance <-> Device 2 (EtherCAT)/Box 1 (AMAX-4870)/Box 51 (BL 570)/DO570 6 (DO 570)
//     Main_IO_Task Inputs/EtherCAT.LoadMod_7.Output_ShortCircuit[{1..16}] <-> DO SC State Mapping/DO{0..15} SC State  (16 links)
//     Main_IO_Task Inputs/EtherCAT.LoadMod_7.State <-> InfoData/State
//     Main_IO_Task Inputs/EtherCAT.LoadMod_7.WcState <-> WcState/WcState
//     Main_IO_Task Outputs/EtherCAT.LoadMod_7.Output[{1..16}] <-> DO Mapping/DO{0..15} Value  (16 links)
//   External_Conveyor_system Instance <-> Device 2 (EtherCAT)/Box 1 (AMAX-4870)/Box 2 (AMAX-4870)/Box 14 (54632)
//     PlcTask Inputs/Sensor.sensor.in_RawData[{0..7}] <-> Module 8 (IOL_8/8_I/O-Bytes)/TxPDO/input byte {0..7}  (8 links)
//     PlcTask Outputs/Sensor.sensor.out_rawdata <-> Module 8 (IOL_8/8_I/O-Bytes)/RxPDO/output byte 0
//   External_Conveyor_system Instance <-> Device 2 (EtherCAT)/Box 1 (AMAX-4870)/Box 51 (BL 570)/Box 53 (MM 540)
//     PlcTask Inputs/Axis.FeedCar_Enc.FeedCar_Enc_raw.Inc <-> Inc Mapping/Inc0 Value
//     PlcTask Inputs/Axis.FeedCar_Enc.FeedCar_Enc_raw.Inc_Error_A <-> Inc Error Mapping/Inc0 Error Track A
//     PlcTask Inputs/Axis.FeedCar_Enc.FeedCar_Enc_raw.Inc_Error_B <-> Inc Error Mapping/Inc0 Error Track B
//     PlcTask Inputs/Axis.FeedCar_Enc.FeedCar_Enc_raw.Inc_Error_C <-> Inc Error Mapping/Inc0 Error 0-Impulse Track
//     PlcTask Inputs/Axis.FeedCar_Enc.FeedCar_Enc_raw.Inc_Preload_Done <-> Inc State Mapping/Inc0 Preload Done
//     PlcTask Outputs/Axis.FeedCar_Enc.FeedCar_Enc_raw.Inc_Preload_Trigger <-> Inc Preload Trigger Mapping/Inc0 Preload Trigger
//     PlcTask Outputs/Axis.FeedCar_Enc.FeedCar_Enc_raw.Inc_Preload_Value <-> Inc Preload Value Mapping/Inc0 Preload Value
//   External_Conveyor_system Instance <-> NC-Task 1 SAF/Axes/轴 19
//     PlcTask Inputs/Axis.Axis_StepMoter.NcToPlc <-> 输出/ToPlc
//     PlcTask Outputs/Axis.Axis_StepMoter.PlcToNc <-> 输入/FromPlc
//   External_Conveyor_system Instance <-> IO_External_Task/IO_External_Task Instance
//     PlcTask Inputs/IO.i101 <-> Main_IO_Task Outputs/MainIO.IO101.In[1]
//     PlcTask Inputs/IO.i102 <-> Main_IO_Task Outputs/MainIO.IO101.In[2]
//     PlcTask Inputs/IO.i103 <-> Main_IO_Task Outputs/MainIO.IO101.In[3]
//     PlcTask Inputs/IO.i104 <-> Main_IO_Task Outputs/MainIO.IO101.In[4]
//     PlcTask Inputs/IO.i105 <-> Main_IO_Task Outputs/MainIO.IO101.In[5]
//     PlcTask Inputs/IO.i106 <-> Main_IO_Task Outputs/MainIO.IO101.In[6]
//     PlcTask Inputs/IO.i107 <-> Main_IO_Task Outputs/MainIO.IO101.In[7]
//     PlcTask Inputs/IO.i108 <-> Main_IO_Task Outputs/MainIO.IO101.In[8]
//     PlcTask Inputs/IO.i109 <-> Main_IO_Task Outputs/MainIO.IO101.In[9]
//     PlcTask Inputs/IO.i110 <-> Main_IO_Task Outputs/MainIO.IO101.In[10]
//     PlcTask Inputs/IO.i111 <-> Main_IO_Task Outputs/MainIO.IO101.In[11]
//     PlcTask Inputs/IO.i112 <-> Main_IO_Task Outputs/MainIO.IO101.In[12]
//     PlcTask Inputs/IO.i113 <-> Main_IO_Task Outputs/MainIO.IO101.In[13]
//     PlcTask Inputs/IO.i114 <-> Main_IO_Task Outputs/MainIO.IO101.In[14]
//     PlcTask Inputs/IO.i115 <-> Main_IO_Task Outputs/MainIO.IO101.In[15]
//     PlcTask Inputs/IO.i116 <-> Main_IO_Task Outputs/MainIO.IO101.In[16]
//     PlcTask Inputs/IO.i201 <-> Main_IO_Task Outputs/MainIO.IO102.In[1]
//     PlcTask Inputs/IO.i202 <-> Main_IO_Task Outputs/MainIO.IO102.In[2]
//     PlcTask Inputs/IO.i203 <-> Main_IO_Task Outputs/MainIO.IO102.In[3]
//     PlcTask Inputs/IO.i204 <-> Main_IO_Task Outputs/MainIO.IO102.In[4]
//     PlcTask Inputs/IO.i205 <-> Main_IO_Task Outputs/MainIO.IO102.In[5]
//     PlcTask Inputs/IO.i206 <-> Main_IO_Task Outputs/MainIO.IO102.In[6]
//     PlcTask Inputs/IO.i207 <-> Main_IO_Task Outputs/MainIO.IO102.In[7]
//     PlcTask Inputs/IO.i208 <-> Main_IO_Task Outputs/MainIO.IO102.In[8]
//     PlcTask Inputs/IO.i209 <-> Main_IO_Task Outputs/MainIO.IO102.In[9]
//     PlcTask Inputs/IO.i210 <-> Main_IO_Task Outputs/MainIO.IO102.In[10]
//     PlcTask Inputs/IO.i211 <-> Main_IO_Task Outputs/MainIO.IO102.In[11]
//     PlcTask Inputs/IO.i212 <-> Main_IO_Task Outputs/MainIO.IO102.In[12]
//     PlcTask Inputs/IO.i213 <-> Main_IO_Task Outputs/MainIO.IO102.In[13]
//     PlcTask Inputs/IO.i214 <-> Main_IO_Task Outputs/MainIO.IO102.In[14]
//     PlcTask Inputs/IO.i215 <-> Main_IO_Task Outputs/MainIO.IO102.In[15]
//     PlcTask Inputs/IO.i216 <-> Main_IO_Task Outputs/MainIO.IO102.In[16]
//     PlcTask Inputs/IO.i301 <-> Main_IO_Task Outputs/MainIO.IO103.In[1]
//     PlcTask Inputs/IO.i302 <-> Main_IO_Task Outputs/MainIO.IO103.In[2]
//     PlcTask Inputs/IO.i303 <-> Main_IO_Task Outputs/MainIO.IO103.In[3]
//     PlcTask Inputs/IO.i304 <-> Main_IO_Task Outputs/MainIO.IO103.In[4]
//     PlcTask Inputs/IO.i305 <-> Main_IO_Task Outputs/MainIO.IO103.In[5]
//     PlcTask Inputs/IO.i306 <-> Main_IO_Task Outputs/MainIO.IO103.In[6]
//     PlcTask Inputs/IO.i307 <-> Main_IO_Task Outputs/MainIO.IO103.In[7]
//     PlcTask Inputs/IO.i308 <-> Main_IO_Task Outputs/MainIO.IO103.In[8]
//     PlcTask Inputs/IO.i309 <-> Main_IO_Task Outputs/MainIO.IO103.In[9]
//     PlcTask Inputs/IO.i310 <-> Main_IO_Task Outputs/MainIO.IO103.In[10]
//     PlcTask Inputs/IO.i311 <-> Main_IO_Task Outputs/MainIO.IO103.In[11]
//     PlcTask Inputs/IO.i312 <-> Main_IO_Task Outputs/MainIO.IO103.In[12]
//     PlcTask Inputs/IO.i313 <-> Main_IO_Task Outputs/MainIO.IO103.In[13]
//     PlcTask Inputs/IO.i314 <-> Main_IO_Task Outputs/MainIO.IO103.In[14]
//     PlcTask Inputs/IO.i315 <-> Main_IO_Task Outputs/MainIO.IO103.In[15]
//     PlcTask Inputs/IO.i316 <-> Main_IO_Task Outputs/MainIO.IO103.In[16]
//     PlcTask Inputs/IO.i401 <-> Main_IO_Task Outputs/MainIO.IO104.In[1]
//     PlcTask Inputs/IO.i402 <-> Main_IO_Task Outputs/MainIO.IO104.In[2]
//     PlcTask Inputs/IO.i403 <-> Main_IO_Task Outputs/MainIO.IO104.In[3]
//     PlcTask Inputs/IO.i404 <-> Main_IO_Task Outputs/MainIO.IO104.In[4]
//     PlcTask Inputs/IO.i405 <-> Main_IO_Task Outputs/MainIO.IO104.In[5]
//     PlcTask Inputs/IO.i406 <-> Main_IO_Task Outputs/MainIO.IO104.In[6]
//     PlcTask Inputs/IO.i407 <-> Main_IO_Task Outputs/MainIO.IO104.In[7]
//     PlcTask Inputs/IO.i408 <-> Main_IO_Task Outputs/MainIO.IO104.In[8]
//     PlcTask Inputs/IO.i409 <-> Main_IO_Task Outputs/MainIO.IO104.In[9]
//     PlcTask Inputs/IO.i410 <-> Main_IO_Task Outputs/MainIO.IO104.In[10]
//     PlcTask Inputs/IO.i411 <-> Main_IO_Task Outputs/MainIO.IO104.In[11]
//     PlcTask Inputs/IO.i412 <-> Main_IO_Task Outputs/MainIO.IO104.In[12]
//     PlcTask Inputs/IO.i413 <-> Main_IO_Task Outputs/MainIO.IO104.In[13]
//     PlcTask Inputs/IO.i414 <-> Main_IO_Task Outputs/MainIO.IO104.In[14]
//     PlcTask Inputs/IO.i415 <-> Main_IO_Task Outputs/MainIO.IO104.In[15]
//     PlcTask Inputs/IO.i416 <-> Main_IO_Task Outputs/MainIO.IO104.In[16]
//     PlcTask Outputs/IO.q101 <-> Main_IO_Task Inputs/MainIO.IO105.Out[1]
//     PlcTask Outputs/IO.q102 <-> Main_IO_Task Inputs/MainIO.IO105.Out[2]
//     PlcTask Outputs/IO.q103 <-> Main_IO_Task Inputs/MainIO.IO105.Out[3]
//     PlcTask Outputs/IO.q104 <-> Main_IO_Task Inputs/MainIO.IO105.Out[4]
//     PlcTask Outputs/IO.q105 <-> Main_IO_Task Inputs/MainIO.IO105.Out[5]
//     PlcTask Outputs/IO.q106 <-> Main_IO_Task Inputs/MainIO.IO105.Out[6]
//     PlcTask Outputs/IO.q107 <-> Main_IO_Task Inputs/MainIO.IO105.Out[7]
//     PlcTask Outputs/IO.q108 <-> Main_IO_Task Inputs/MainIO.IO105.Out[8]
//     PlcTask Outputs/IO.q109 <-> Main_IO_Task Inputs/MainIO.IO105.Out[9]
//     PlcTask Outputs/IO.q110 <-> Main_IO_Task Inputs/MainIO.IO105.Out[10]
//     PlcTask Outputs/IO.q111 <-> Main_IO_Task Inputs/MainIO.IO105.Out[11]
//     PlcTask Outputs/IO.q112 <-> Main_IO_Task Inputs/MainIO.IO105.Out[12]
//     PlcTask Outputs/IO.q113 <-> Main_IO_Task Inputs/MainIO.IO105.Out[13]
//     PlcTask Outputs/IO.q114 <-> Main_IO_Task Inputs/MainIO.IO105.Out[14]
//     PlcTask Outputs/IO.q115 <-> Main_IO_Task Inputs/MainIO.IO105.Out[15]
//     PlcTask Outputs/IO.q116 <-> Main_IO_Task Inputs/MainIO.IO105.Out[16]
//     PlcTask Outputs/IO.q201 <-> Main_IO_Task Inputs/MainIO.IO106.Out[1]
//     PlcTask Outputs/IO.q202 <-> Main_IO_Task Inputs/MainIO.IO106.Out[2]
//     PlcTask Outputs/IO.q203 <-> Main_IO_Task Inputs/MainIO.IO106.Out[3]
//     PlcTask Outputs/IO.q204 <-> Main_IO_Task Inputs/MainIO.IO106.Out[4]
//     PlcTask Outputs/IO.q205 <-> Main_IO_Task Inputs/MainIO.IO106.Out[5]
//     PlcTask Outputs/IO.q206 <-> Main_IO_Task Inputs/MainIO.IO106.Out[6]
//     PlcTask Outputs/IO.q207 <-> Main_IO_Task Inputs/MainIO.IO106.Out[7]
//     PlcTask Outputs/IO.q208 <-> Main_IO_Task Inputs/MainIO.IO106.Out[8]
//     PlcTask Outputs/IO.q209 <-> Main_IO_Task Inputs/MainIO.IO106.Out[9]
//     PlcTask Outputs/IO.q210 <-> Main_IO_Task Inputs/MainIO.IO106.Out[10]
//     PlcTask Outputs/IO.q211 <-> Main_IO_Task Inputs/MainIO.IO106.Out[11]
//     PlcTask Outputs/IO.q212 <-> Main_IO_Task Inputs/MainIO.IO106.Out[12]
//     PlcTask Outputs/IO.q213 <-> Main_IO_Task Inputs/MainIO.IO106.Out[13]
//     PlcTask Outputs/IO.q214 <-> Main_IO_Task Inputs/MainIO.IO106.Out[14]
//     PlcTask Outputs/IO.q215 <-> Main_IO_Task Inputs/MainIO.IO106.Out[15]
//     PlcTask Outputs/IO.q216 <-> Main_IO_Task Inputs/MainIO.IO106.Out[16]
//     PlcTask Outputs/IO.q301 <-> Main_IO_Task Inputs/MainIO.IO107.Out[1]
//     PlcTask Outputs/IO.q302 <-> Main_IO_Task Inputs/MainIO.IO107.Out[2]
//     PlcTask Outputs/IO.q303 <-> Main_IO_Task Inputs/MainIO.IO107.Out[3]
//     PlcTask Outputs/IO.q304 <-> Main_IO_Task Inputs/MainIO.IO107.Out[4]
//     PlcTask Outputs/IO.q305 <-> Main_IO_Task Inputs/MainIO.IO107.Out[5]
//     PlcTask Outputs/IO.q306 <-> Main_IO_Task Inputs/MainIO.IO107.Out[6]
//     PlcTask Outputs/IO.q307 <-> Main_IO_Task Inputs/MainIO.IO107.Out[7]
//     PlcTask Outputs/IO.q308 <-> Main_IO_Task Inputs/MainIO.IO107.Out[8]
//     PlcTask Outputs/IO.q309 <-> Main_IO_Task Inputs/MainIO.IO107.Out[9]
//     PlcTask Outputs/IO.q310 <-> Main_IO_Task Inputs/MainIO.IO107.Out[10]
//     PlcTask Outputs/IO.q311 <-> Main_IO_Task Inputs/MainIO.IO107.Out[11]
//     PlcTask Outputs/IO.q312 <-> Main_IO_Task Inputs/MainIO.IO107.Out[12]
//     PlcTask Outputs/IO.q313 <-> Main_IO_Task Inputs/MainIO.IO107.Out[13]
//     PlcTask Outputs/IO.q314 <-> Main_IO_Task Inputs/MainIO.IO107.Out[14]
//     PlcTask Outputs/IO.q315 <-> Main_IO_Task Inputs/MainIO.IO107.Out[15]
//     PlcTask Outputs/IO.q316 <-> Main_IO_Task Inputs/MainIO.IO107.Out[16]
//   External_Conveyor_system Instance <-> Main/Main Instance
//     PlcTask Inputs/Input.Feed_Enable <-> PlcTask Outputs/ExpConver.ExpConver_Enable
//     PlcTask Inputs/Input.Feed_Mode <-> PlcTask Outputs/ExpConver.ExpConver_Mode
//     PlcTask Inputs/Input.Feed_Reset <-> PlcTask Outputs/ExpConver.ExpConver_Reset
//     PlcTask Inputs/Input.Feed_Start <-> PlcTask Outputs/ExpConver.ExpConver_Start
//     PlcTask Inputs/Input.Feed_WorkOrder_UUID <-> PlcTask Outputs/ExpConver.ExpConver_WorkOrder_UUID
//     PlcTask Inputs/Input.In_Moter_Start <-> PlcTask Outputs/ExpConver.In_Moter_Start
//     PlcTask Inputs/Input.Out_Moter_Start <-> PlcTask Outputs/ExpConver.Out_Moter_Start
//     PlcTask Inputs/Input.PullOver_Start <-> PlcTask Outputs/ExpConver.PullOver_Start
//     PlcTask Outputs/Output.ActionMode_Now <-> PlcTask Inputs/ExpConver.ActionMode_Now
//     PlcTask Outputs/Output.Feed_Workpiace_H <-> PlcTask Inputs/ExpConver.Feed_Workpiace_H
//     PlcTask Outputs/Output.Feed_Workpiace_W <-> PlcTask Inputs/ExpConver.Feed_Workpiace_W
//     PlcTask Outputs/Output.Feed_bBuzy <-> PlcTask Inputs/ExpConver.Feed_bBuzy
//     PlcTask Outputs/Output.Feed_bDone <-> PlcTask Inputs/ExpConver.Feed_bDone
//     PlcTask Outputs/Output.Feed_bError <-> PlcTask Inputs/ExpConver.Feed_bError
//     PlcTask Outputs/Output.In_Moter_Error <-> PlcTask Inputs/ExpConver.In_Moter_Error
//     PlcTask Outputs/Output.In_Moter_Running <-> PlcTask Inputs/ExpConver.In_Moter_Running
